// TwinCAT 3 PLC project LeakTesters
// ProgramVersion: 3.1.4024.0
// libraries:
//   Tc2_Standard, * (Beckhoff Automation GmbH)
//   Tc2_System, * (Beckhoff Automation GmbH)
//   Tc2_Utilities, * (Beckhoff Automation GmbH)
//   Tc3_EventLogger, * (Beckhoff Automation GmbH)
//   Tc3_Module, * (Beckhoff Automation GmbH)
//   VisuUserMgmt, * (System)
// project tree:
//   DUTs/ E_CameraJobChange.TcDUT, E_MachineState.TcDUT (not stored), E_StationState.TcDUT (not stored), ST_ActiveEventsHMI.TcDUT (not stored), ST_AlarmHistory.TcDUT (not stored), ST_Events.TcDUT (not stored), ST_HeightLimits.TcDUT, ST_HeightMeasurement2.TcDUT, ST_MachineStatusStruct.TcDUT (not stored), ST_MasterControlStruct.TcDUT (not stored), ST_MeasureStatistics.TcDUT (not stored), ST_Nest.TcDUT, ST_PartsInspection.TcDUT, ST_StandardStationStruct.TcDUT (not stored), ST_UserLogHMI.TcDUT (not stored)
//   DUTs/HeightMeasureFunction/ E_HeighttMeasureProcess.TcDUT
//   DUTs/IO/i28/ st_i28General_I_O.TcDUT (not stored), st_i28LasResult.TcDUT (not stored), st_i28LiveMeasurement.TcDUT (not stored)
//   DUTs/IO/ st_IS2802M.TcDUT, E_BoxDiag.TcDUT (not stored), E_BoxState.TcDUT (not stored), E_TerminalState.TcDUT (not stored), st_Box_Info.TcDUT (not stored), st_EL1809.TcDUT (not stored), st_EL2809.TcDUT (not stored), ST_DL_PN1.TcDUT, st_Terminal_Info.TcDUT (not stored)
//   GVLs/ GVL_Constants.TcGVL (not stored), GVL_HMI_GLOBAL.TcGVL, GVL_IO.TcGVL, GVL_MASTER.TcGVL, GVL_PERSIST.TcGVL
//   / PlcTask.TcTTO (not stored)
//   POUs/A_Master/ Main_Master.TcPOU, PRG_FaultHandling.TcPOU, PRG_MachineStatus.TcPOU, PRG_MasterCycle.TcPOU, PRG_MasterSystemTime.TcPOU (not stored), PRG_TerminBoxInfo.TcPOU (not stored)
//   POUs/B_HightTest/ PRG_Fault_HeightTest.TcPOU, PRG_HeightTest.TcPOU
//   POUs/C_LeakTest/ PRG_Fault_LeakTest.TcPOU, PRG_LeakTest.TcPOU, PRG_LeakTestEvents_Info.TcPOU
//   POUs/D_VisionTest/ PRG_Fault_VisionTest.TcPOU, PRG_VisionTest.TcPOU
//   POUs/E_HMI/ PRG_HMI.TcPOU
//   POUs/G_Utility/ FB_Alarms.TcPOU (not stored), FB_BoxInfo.TcPOU (not stored), FB_DayOfYear.TcPOU (not stored), FB_EventLog.TcPOU (not stored), FB_HeightMeasurement2.TcPOU, FB_Pulse.TcPOU (not stored), FB_TerminalInfo.TcPOU (not stored), FB_TimeControl.TcPOU (not stored), PRG_Puls.TcPOU (not stored)
//   POUs/ MAIN.TcPOU (not stored)
// real-time tasks:
//   TASK PlcTask: cycle T#10ms, priority 20, ADS port 350
// I/O:
//   DEVICE Device 1 (EtherCAT), AmsNetId 172.18.237.82.2.1
//     Term 9 (EK1100) [EK1100 EtherCAT Coupler (2A E-Bus)]
//       Term 10 (EL6070-0033) [EL6070-0033 1Ch. Licence key terminal, individual licences]
//       Term 11 (EL1809) [EL1809 16Ch. Dig. Input 24V, 3ms]
//       Term 12 (EL2809-0015) [EL2809-0015 16Ch. Dig. Output 24V DC, 0.35A, not short-circuit proof]
//       Term 13 (EL6631) [EL6631 PROFINET IO Controller]
//       Term 14 (EL9011) [EL9011 End Terminal]
//   DEVICE Device 2 (EL6631), AmsNetId 172.18.237.82.3.1
//     is2802 [Cognex Corp. In-Sight IS28XX Vision System IS28XX-XX]
//       modules: Term 1 (DAP Module), Term 2 (Acquisition Control), Term 3 (Acquisition Status), Term 4 (Inspection Control), Term 5 (Inspection Status), Term 6 (Command Control), Term 7 (ExternalEvent Control), Term 8 (User Data - 64 bytes), Term 9 (Results - 64 bytes)
//     i28 [Cincinnati Test Systems 1-port Device 00210]
//       modules: Term 10 (DAP Module), Term 11 (PLC Input), Term 12 (PLC Output  )
//     dl-pn1 [Keyence DL-PN1 PROFINET IO Device DL-PN1]
//       modules: Term 13 (DAP Module), Term 14 (DL-PN1), Term 15 (GT2-1.1), Term 16 (GT2-1.2), Term 17 (GT2-1.3), Term 18 (GT2-2)
// variable links:
//   LeakTesters/LeakTesters Instance <-> Device 1 (EtherCAT)/Term 9 (EK1100)/Term 10 (EL6070-0033)
//     PlcTask Inputs/GVL_IO.dwTerminalInfo[2].nTerminal_State <-> InfoData/State
//   LeakTesters/LeakTesters Instance <-> Device 1 (EtherCAT)/Term 9 (EK1100)/Term 11 (EL1809)
//     PlcTask Inputs/GVL_IO.dwTerminalInfo[3].nTerminal_State <-> InfoData/State
//     PlcTask Inputs/GVL_IO.dw_T02_EL1809.iCalmpClosed <-> Channel 1/Input
//     PlcTask Inputs/GVL_IO.dw_T02_EL1809.iPartPresent <-> Channel 2/Input
//   LeakTesters/LeakTesters Instance <-> Device 1 (EtherCAT)/Term 9 (EK1100)/Term 12 (EL2809-0015)
//     PlcTask Inputs/GVL_IO.dwTerminalInfo[4].nTerminal_State <-> InfoData/State
//     PlcTask Outputs/GVL_IO.dw_T03_EL2809.qEL2809_Ch3 <-> Channel 3/Output
//     PlcTask Outputs/GVL_IO.dw_T03_EL2809.qPassIndicatorGreen <-> Channel 1/Output
//     PlcTask Outputs/GVL_IO.dw_T03_EL2809.qRejectIndicatorRed <-> Channel 2/Output
//   LeakTesters/LeakTesters Instance <-> Device 1 (EtherCAT)/Term 9 (EK1100)/Term 13 (EL6631)
//     PlcTask Inputs/GVL_IO.dwTerminalInfo[5].nTerminal_State <-> InfoData/State
//   LeakTesters/LeakTesters Instance <-> Device 2 (EL6631)/dl-pn1
//     PlcTask Inputs/GVL_IO.dwBoxInfo[17].nPnIoBoxDiag <-> Inputs/PnIoBoxDiag
//     PlcTask Inputs/GVL_IO.dwBoxInfo[17].nPnIoBoxState <-> Inputs/PnIoBoxState
//     PlcTask Inputs/GVL_IO.dw_B08_DL_PN1.dldCurrValProp <-> API/Term 14 (DL-PN1)/Subterm 23 (DL-PN1 Device)/Inputs/Sensors Status/Current_Value_Property
//     PlcTask Inputs/GVL_IO.dw_B08_DL_PN1.dldErrorStt <-> API/Term 14 (DL-PN1)/Subterm 23 (DL-PN1 Device)/Inputs/Sensors Status/Error_Status
//     PlcTask Inputs/GVL_IO.dw_B08_DL_PN1.dldExtInpResp[1] <-> API/Term 14 (DL-PN1)/Subterm 23 (DL-PN1 Device)/Inputs/External Input Response/External_Input_Response_1
//     PlcTask Inputs/GVL_IO.dw_B08_DL_PN1.dldExtInpResp[2] <-> API/Term 14 (DL-PN1)/Subterm 23 (DL-PN1 Device)/Inputs/External Input Response/External_Input_Response_2
//     PlcTask Inputs/GVL_IO.dw_B08_DL_PN1.dldExtInpResp[3] <-> API/Term 14 (DL-PN1)/Subterm 23 (DL-PN1 Device)/Inputs/External Input Response/External_Input_Response_3
//     PlcTask Inputs/GVL_IO.dw_B08_DL_PN1.dldExtInpResp[4] <-> API/Term 14 (DL-PN1)/Subterm 23 (DL-PN1 Device)/Inputs/External Input Response/External_Input_Response_4
//     PlcTask Inputs/GVL_IO.dw_B08_DL_PN1.dldExtInpResp[5] <-> API/Term 14 (DL-PN1)/Subterm 23 (DL-PN1 Device)/Inputs/External Input Response/External_Input_Response_5
//     PlcTask Inputs/GVL_IO.dw_B08_DL_PN1.dldWarningStat <-> API/Term 14 (DL-PN1)/Subterm 23 (DL-PN1 Device)/Inputs/Sensors Status/Warning_Status
//     PlcTask Inputs/GVL_IO.dw_B08_DL_PN1.gt2_1_1CurrValInv <-> API/Term 15 (GT2-1.1)/Subterm 24 (GT2-***)/Inputs/Sensor Status/Current_Value_Invalid
//     PlcTask Inputs/GVL_IO.dw_B08_DL_PN1.gt2_1_2CurrValInv <-> API/Term 16 (GT2-1.2)/Subterm 25 (GT2-***)/Inputs/Sensor Status/Current_Value_Invalid
//     PlcTask Inputs/GVL_IO.dw_B08_DL_PN1.gt2_1_3CurrValInv <-> API/Term 17 (GT2-1.3)/Subterm 26 (GT2-***)/Inputs/Sensor Status/Current_Value_Invalid
//     PlcTask Inputs/GVL_IO.dw_B08_DL_PN1.gt2_1_1CurrValOvrR <-> API/Term 15 (GT2-1.1)/Subterm 24 (GT2-***)/Inputs/Sensor Status/Current_Value_Over_Range
//     PlcTask Inputs/GVL_IO.dw_B08_DL_PN1.gt2_1_2CurrValOvrR <-> API/Term 16 (GT2-1.2)/Subterm 25 (GT2-***)/Inputs/Sensor Status/Current_Value_Over_Range
//     PlcTask Inputs/GVL_IO.dw_B08_DL_PN1.gt2_1_3CurrValOvrR <-> API/Term 17 (GT2-1.3)/Subterm 26 (GT2-***)/Inputs/Sensor Status/Current_Value_Over_Range
//     PlcTask Inputs/GVL_IO.dw_B08_DL_PN1.gt2_1_1CurrValUndR <-> API/Term 15 (GT2-1.1)/Subterm 24 (GT2-***)/Inputs/Sensor Status/Current_Value_Under_Range
//     PlcTask Inputs/GVL_IO.dw_B08_DL_PN1.gt2_1_2CurrValUndR <-> API/Term 16 (GT2-1.2)/Subterm 25 (GT2-***)/Inputs/Sensor Status/Current_Value_Under_Range
//     PlcTask Inputs/GVL_IO.dw_B08_DL_PN1.gt2_1_3CurrValUndR <-> API/Term 17 (GT2-1.3)/Subterm 26 (GT2-***)/Inputs/Sensor Status/Current_Value_Under_Range
//     PlcTask Inputs/GVL_IO.dw_B08_DL_PN1.gt2_1_1CurrentValue <-> API/Term 15 (GT2-1.1)/Subterm 24 (GT2-***)/Inputs/Current Value
//     PlcTask Inputs/GVL_IO.dw_B08_DL_PN1.gt2_1_2CurrentValue <-> API/Term 16 (GT2-1.2)/Subterm 25 (GT2-***)/Inputs/Current Value
//     PlcTask Inputs/GVL_IO.dw_B08_DL_PN1.gt2_1_3CurrentValue <-> API/Term 17 (GT2-1.3)/Subterm 26 (GT2-***)/Inputs/Current Value
//     PlcTask Inputs/GVL_IO.dw_B08_DL_PN1.gt2_1_1ErrorStat <-> API/Term 15 (GT2-1.1)/Subterm 24 (GT2-***)/Inputs/Sensor Status/Error_Status
//     PlcTask Inputs/GVL_IO.dw_B08_DL_PN1.gt2_1_2ErrorStat <-> API/Term 16 (GT2-1.2)/Subterm 25 (GT2-***)/Inputs/Sensor Status/Error_Status
//     PlcTask Inputs/GVL_IO.dw_B08_DL_PN1.gt2_1_3ErrorStat <-> API/Term 17 (GT2-1.3)/Subterm 26 (GT2-***)/Inputs/Sensor Status/Error_Status
//     PlcTask Inputs/GVL_IO.dw_B08_DL_PN1.gt2_1_1ExtInpRes[1] <-> API/Term 15 (GT2-1.1)/Subterm 24 (GT2-***)/Inputs/External Input Response/External_Input_Response_1
//     PlcTask Inputs/GVL_IO.dw_B08_DL_PN1.gt2_1_1ExtInpRes[2] <-> API/Term 15 (GT2-1.1)/Subterm 24 (GT2-***)/Inputs/External Input Response/External_Input_Response_2
//     PlcTask Inputs/GVL_IO.dw_B08_DL_PN1.gt2_1_1ExtInpRes[3] <-> API/Term 15 (GT2-1.1)/Subterm 24 (GT2-***)/Inputs/External Input Response/External_Input_Response_3
//     PlcTask Inputs/GVL_IO.dw_B08_DL_PN1.gt2_1_1ExtInpRes[4] <-> API/Term 15 (GT2-1.1)/Subterm 24 (GT2-***)/Inputs/External Input Response/External_Input_Response_4
//     PlcTask Inputs/GVL_IO.dw_B08_DL_PN1.gt2_1_1ExtInpRes[5] <-> API/Term 15 (GT2-1.1)/Subterm 24 (GT2-***)/Inputs/External Input Response/External_Input_Response_5
//     PlcTask Inputs/GVL_IO.dw_B08_DL_PN1.gt2_1_2ExtInpRes[1] <-> API/Term 16 (GT2-1.2)/Subterm 25 (GT2-***)/Inputs/External Input Response/External_Input_Response_1
//     PlcTask Inputs/GVL_IO.dw_B08_DL_PN1.gt2_1_2ExtInpRes[2] <-> API/Term 16 (GT2-1.2)/Subterm 25 (GT2-***)/Inputs/External Input Response/External_Input_Response_2
//     PlcTask Inputs/GVL_IO.dw_B08_DL_PN1.gt2_1_2ExtInpRes[3] <-> API/Term 16 (GT2-1.2)/Subterm 25 (GT2-***)/Inputs/External Input Response/External_Input_Response_3
//     PlcTask Inputs/GVL_IO.dw_B08_DL_PN1.gt2_1_2ExtInpRes[4] <-> API/Term 16 (GT2-1.2)/Subterm 25 (GT2-***)/Inputs/External Input Response/External_Input_Response_4
//     PlcTask Inputs/GVL_IO.dw_B08_DL_PN1.gt2_1_2ExtInpRes[5] <-> API/Term 16 (GT2-1.2)/Subterm 25 (GT2-***)/Inputs/External Input Response/External_Input_Response_5
//     PlcTask Inputs/GVL_IO.dw_B08_DL_PN1.gt2_1_3ExtInpRes[1] <-> API/Term 17 (GT2-1.3)/Subterm 26 (GT2-***)/Inputs/External Input Response/External_Input_Response_1
//     PlcTask Inputs/GVL_IO.dw_B08_DL_PN1.gt2_1_3ExtInpRes[2] <-> API/Term 17 (GT2-1.3)/Subterm 26 (GT2-***)/Inputs/External Input Response/External_Input_Response_2
//     PlcTask Inputs/GVL_IO.dw_B08_DL_PN1.gt2_1_3ExtInpRes[3] <-> API/Term 17 (GT2-1.3)/Subterm 26 (GT2-***)/Inputs/External Input Response/External_Input_Response_3
//     PlcTask Inputs/GVL_IO.dw_B08_DL_PN1.gt2_1_3ExtInpRes[4] <-> API/Term 17 (GT2-1.3)/Subterm 26 (GT2-***)/Inputs/External Input Response/External_Input_Response_4
//     PlcTask Inputs/GVL_IO.dw_B08_DL_PN1.gt2_1_3ExtInpRes[5] <-> API/Term 17 (GT2-1.3)/Subterm 26 (GT2-***)/Inputs/External Input Response/External_Input_Response_5
//     PlcTask Inputs/GVL_IO.dw_B08_DL_PN1.gt2_1_1Output[1] <-> API/Term 15 (GT2-1.1)/Subterm 24 (GT2-***)/Inputs/Sensor Outputs/Output_1
//     PlcTask Inputs/GVL_IO.dw_B08_DL_PN1.gt2_1_1Output[2] <-> API/Term 15 (GT2-1.1)/Subterm 24 (GT2-***)/Inputs/Sensor Outputs/Output_2
//     PlcTask Inputs/GVL_IO.dw_B08_DL_PN1.gt2_1_1Output[3] <-> API/Term 15 (GT2-1.1)/Subterm 24 (GT2-***)/Inputs/Sensor Outputs/Output_3
//     PlcTask Inputs/GVL_IO.dw_B08_DL_PN1.gt2_1_1Output[4] <-> API/Term 15 (GT2-1.1)/Subterm 24 (GT2-***)/Inputs/Sensor Outputs/Output_4
//     PlcTask Inputs/GVL_IO.dw_B08_DL_PN1.gt2_1_1Output[5] <-> API/Term 15 (GT2-1.1)/Subterm 24 (GT2-***)/Inputs/Sensor Outputs/Output_5
//     PlcTask Inputs/GVL_IO.dw_B08_DL_PN1.gt2_1_2Output[1] <-> API/Term 16 (GT2-1.2)/Subterm 25 (GT2-***)/Inputs/Sensor Outputs/Output_1
//     PlcTask Inputs/GVL_IO.dw_B08_DL_PN1.gt2_1_2Output[2] <-> API/Term 16 (GT2-1.2)/Subterm 25 (GT2-***)/Inputs/Sensor Outputs/Output_2
//     PlcTask Inputs/GVL_IO.dw_B08_DL_PN1.gt2_1_2Output[3] <-> API/Term 16 (GT2-1.2)/Subterm 25 (GT2-***)/Inputs/Sensor Outputs/Output_3
//     PlcTask Inputs/GVL_IO.dw_B08_DL_PN1.gt2_1_2Output[4] <-> API/Term 16 (GT2-1.2)/Subterm 25 (GT2-***)/Inputs/Sensor Outputs/Output_4
//     PlcTask Inputs/GVL_IO.dw_B08_DL_PN1.gt2_1_2Output[5] <-> API/Term 16 (GT2-1.2)/Subterm 25 (GT2-***)/Inputs/Sensor Outputs/Output_5
//     PlcTask Inputs/GVL_IO.dw_B08_DL_PN1.gt2_1_3Output[1] <-> API/Term 17 (GT2-1.3)/Subterm 26 (GT2-***)/Inputs/Sensor Outputs/Output_1
//     PlcTask Inputs/GVL_IO.dw_B08_DL_PN1.gt2_1_3Output[2] <-> API/Term 17 (GT2-1.3)/Subterm 26 (GT2-***)/Inputs/Sensor Outputs/Output_2
//     PlcTask Inputs/GVL_IO.dw_B08_DL_PN1.gt2_1_3Output[3] <-> API/Term 17 (GT2-1.3)/Subterm 26 (GT2-***)/Inputs/Sensor Outputs/Output_3
//     PlcTask Inputs/GVL_IO.dw_B08_DL_PN1.gt2_1_3Output[4] <-> API/Term 17 (GT2-1.3)/Subterm 26 (GT2-***)/Inputs/Sensor Outputs/Output_4
//     PlcTask Inputs/GVL_IO.dw_B08_DL_PN1.gt2_1_3Output[5] <-> API/Term 17 (GT2-1.3)/Subterm 26 (GT2-***)/Inputs/Sensor Outputs/Output_5
//     PlcTask Inputs/GVL_IO.dw_B08_DL_PN1.gt2_1_1WarningStat <-> API/Term 15 (GT2-1.1)/Subterm 24 (GT2-***)/Inputs/Sensor Status/Warning_Status
//     PlcTask Inputs/GVL_IO.dw_B08_DL_PN1.gt2_1_2WarningStat <-> API/Term 16 (GT2-1.2)/Subterm 25 (GT2-***)/Inputs/Sensor Status/Warning_Status
//     PlcTask Inputs/GVL_IO.dw_B08_DL_PN1.gt2_1_3WarningStat <-> API/Term 17 (GT2-1.3)/Subterm 26 (GT2-***)/Inputs/Sensor Status/Warning_Status
//     PlcTask Inputs/GVL_IO.dw_B08_DL_PN1.gt2_2CurrValInv <-> API/Term 18 (GT2-2)/Subterm 27 (GT2-***)/Inputs/Sensor Status/Current_Value_Invalid
//     PlcTask Inputs/GVL_IO.dw_B08_DL_PN1.gt2_2CurrValOvrR <-> API/Term 18 (GT2-2)/Subterm 27 (GT2-***)/Inputs/Sensor Status/Current_Value_Over_Range
//     PlcTask Inputs/GVL_IO.dw_B08_DL_PN1.gt2_2CurrValUndR <-> API/Term 18 (GT2-2)/Subterm 27 (GT2-***)/Inputs/Sensor Status/Current_Value_Under_Range
//     PlcTask Inputs/GVL_IO.dw_B08_DL_PN1.gt2_2CurrentValue <-> API/Term 18 (GT2-2)/Subterm 27 (GT2-***)/Inputs/Current Value
//     PlcTask Inputs/GVL_IO.dw_B08_DL_PN1.gt2_2ErrorStat <-> API/Term 18 (GT2-2)/Subterm 27 (GT2-***)/Inputs/Sensor Status/Error_Status
//     PlcTask Inputs/GVL_IO.dw_B08_DL_PN1.gt2_2ExtInpRes[1] <-> API/Term 18 (GT2-2)/Subterm 27 (GT2-***)/Inputs/External Input Response/External_Input_Response_1
//     PlcTask Inputs/GVL_IO.dw_B08_DL_PN1.gt2_2ExtInpRes[2] <-> API/Term 18 (GT2-2)/Subterm 27 (GT2-***)/Inputs/External Input Response/External_Input_Response_2
//     PlcTask Inputs/GVL_IO.dw_B08_DL_PN1.gt2_2ExtInpRes[3] <-> API/Term 18 (GT2-2)/Subterm 27 (GT2-***)/Inputs/External Input Response/External_Input_Response_3
//     PlcTask Inputs/GVL_IO.dw_B08_DL_PN1.gt2_2ExtInpRes[4] <-> API/Term 18 (GT2-2)/Subterm 27 (GT2-***)/Inputs/External Input Response/External_Input_Response_4
//     PlcTask Inputs/GVL_IO.dw_B08_DL_PN1.gt2_2ExtInpRes[5] <-> API/Term 18 (GT2-2)/Subterm 27 (GT2-***)/Inputs/External Input Response/External_Input_Response_5
//     PlcTask Inputs/GVL_IO.dw_B08_DL_PN1.gt2_2Output[1] <-> API/Term 18 (GT2-2)/Subterm 27 (GT2-***)/Inputs/Sensor Outputs/Output_1
//     PlcTask Inputs/GVL_IO.dw_B08_DL_PN1.gt2_2Output[2] <-> API/Term 18 (GT2-2)/Subterm 27 (GT2-***)/Inputs/Sensor Outputs/Output_2
//     PlcTask Inputs/GVL_IO.dw_B08_DL_PN1.gt2_2Output[3] <-> API/Term 18 (GT2-2)/Subterm 27 (GT2-***)/Inputs/Sensor Outputs/Output_3
//     PlcTask Inputs/GVL_IO.dw_B08_DL_PN1.gt2_2Output[4] <-> API/Term 18 (GT2-2)/Subterm 27 (GT2-***)/Inputs/Sensor Outputs/Output_4
//     PlcTask Inputs/GVL_IO.dw_B08_DL_PN1.gt2_2Output[5] <-> API/Term 18 (GT2-2)/Subterm 27 (GT2-***)/Inputs/Sensor Outputs/Output_5
//     PlcTask Inputs/GVL_IO.dw_B08_DL_PN1.gt2_2WarningStat <-> API/Term 18 (GT2-2)/Subterm 27 (GT2-***)/Inputs/Sensor Status/Warning_Status
//     PlcTask Outputs/GVL_IO.dw_B08_DL_PN1.dldExtInpRespOut[1] <-> API/Term 14 (DL-PN1)/Subterm 23 (DL-PN1 Device)/Outputs/External Input Requests/External_Input_Request_1
//     PlcTask Outputs/GVL_IO.dw_B08_DL_PN1.dldExtInpRespOut[2] <-> API/Term 14 (DL-PN1)/Subterm 23 (DL-PN1 Device)/Outputs/External Input Requests/External_Input_Request_2
//     PlcTask Outputs/GVL_IO.dw_B08_DL_PN1.dldExtInpRespOut[3] <-> API/Term 14 (DL-PN1)/Subterm 23 (DL-PN1 Device)/Outputs/External Input Requests/External_Input_Request_3
//     PlcTask Outputs/GVL_IO.dw_B08_DL_PN1.dldExtInpRespOut[4] <-> API/Term 14 (DL-PN1)/Subterm 23 (DL-PN1 Device)/Outputs/External Input Requests/External_Input_Request_4
//     PlcTask Outputs/GVL_IO.dw_B08_DL_PN1.dldExtInpRespOut[5] <-> API/Term 14 (DL-PN1)/Subterm 23 (DL-PN1 Device)/Outputs/External Input Requests/External_Input_Request_5
//     PlcTask Outputs/GVL_IO.dw_B08_DL_PN1.gt2_1_1ExtInpResOut[1] <-> API/Term 15 (GT2-1.1)/Subterm 24 (GT2-***)/Outputs/External Input Requests/External_Input_Request_1
//     PlcTask Outputs/GVL_IO.dw_B08_DL_PN1.gt2_1_1ExtInpResOut[2] <-> API/Term 15 (GT2-1.1)/Subterm 24 (GT2-***)/Outputs/External Input Requests/External_Input_Request_2
//     PlcTask Outputs/GVL_IO.dw_B08_DL_PN1.gt2_1_1ExtInpResOut[3] <-> API/Term 15 (GT2-1.1)/Subterm 24 (GT2-***)/Outputs/External Input Requests/External_Input_Request_3
//     PlcTask Outputs/GVL_IO.dw_B08_DL_PN1.gt2_1_1ExtInpResOut[4] <-> API/Term 15 (GT2-1.1)/Subterm 24 (GT2-***)/Outputs/External Input Requests/External_Input_Request_4
//     PlcTask Outputs/GVL_IO.dw_B08_DL_PN1.gt2_1_1ExtInpResOut[5] <-> API/Term 15 (GT2-1.1)/Subterm 24 (GT2-***)/Outputs/External Input Requests/External_Input_Request_5
//     PlcTask Outputs/GVL_IO.dw_B08_DL_PN1.gt2_1_2ExtInpResOut[1] <-> API/Term 16 (GT2-1.2)/Subterm 25 (GT2-***)/Outputs/External Input Requests/External_Input_Request_1
//     PlcTask Outputs/GVL_IO.dw_B08_DL_PN1.gt2_1_2ExtInpResOut[2] <-> API/Term 16 (GT2-1.2)/Subterm 25 (GT2-***)/Outputs/External Input Requests/External_Input_Request_2
//     PlcTask Outputs/GVL_IO.dw_B08_DL_PN1.gt2_1_2ExtInpResOut[3] <-> API/Term 16 (GT2-1.2)/Subterm 25 (GT2-***)/Outputs/External Input Requests/External_Input_Request_3
//     PlcTask Outputs/GVL_IO.dw_B08_DL_PN1.gt2_1_2ExtInpResOut[4] <-> API/Term 16 (GT2-1.2)/Subterm 25 (GT2-***)/Outputs/External Input Requests/External_Input_Request_4
//     PlcTask Outputs/GVL_IO.dw_B08_DL_PN1.gt2_1_2ExtInpResOut[5] <-> API/Term 16 (GT2-1.2)/Subterm 25 (GT2-***)/Outputs/External Input Requests/External_Input_Request_5
//     PlcTask Outputs/GVL_IO.dw_B08_DL_PN1.gt2_1_3ExtInpResOut[1] <-> API/Term 17 (GT2-1.3)/Subterm 26 (GT2-***)/Outputs/External Input Requests/External_Input_Request_1
//     PlcTask Outputs/GVL_IO.dw_B08_DL_PN1.gt2_1_3ExtInpResOut[2] <-> API/Term 17 (GT2-1.3)/Subterm 26 (GT2-***)/Outputs/External Input Requests/External_Input_Request_2
//     PlcTask Outputs/GVL_IO.dw_B08_DL_PN1.gt2_1_3ExtInpResOut[3] <-> API/Term 17 (GT2-1.3)/Subterm 26 (GT2-***)/Outputs/External Input Requests/External_Input_Request_3
//     PlcTask Outputs/GVL_IO.dw_B08_DL_PN1.gt2_1_3ExtInpResOut[4] <-> API/Term 17 (GT2-1.3)/Subterm 26 (GT2-***)/Outputs/External Input Requests/External_Input_Request_4
//     PlcTask Outputs/GVL_IO.dw_B08_DL_PN1.gt2_1_3ExtInpResOut[5] <-> API/Term 17 (GT2-1.3)/Subterm 26 (GT2-***)/Outputs/External Input Requests/External_Input_Request_5
//     PlcTask Outputs/GVL_IO.dw_B08_DL_PN1.gt2_2ExtInpResOut[1] <-> API/Term 18 (GT2-2)/Subterm 27 (GT2-***)/Outputs/External Input Requests/External_Input_Request_1
//     PlcTask Outputs/GVL_IO.dw_B08_DL_PN1.gt2_2ExtInpResOut[2] <-> API/Term 18 (GT2-2)/Subterm 27 (GT2-***)/Outputs/External Input Requests/External_Input_Request_2
//     PlcTask Outputs/GVL_IO.dw_B08_DL_PN1.gt2_2ExtInpResOut[3] <-> API/Term 18 (GT2-2)/Subterm 27 (GT2-***)/Outputs/External Input Requests/External_Input_Request_3
//     PlcTask Outputs/GVL_IO.dw_B08_DL_PN1.gt2_2ExtInpResOut[4] <-> API/Term 18 (GT2-2)/Subterm 27 (GT2-***)/Outputs/External Input Requests/External_Input_Request_4
//     PlcTask Outputs/GVL_IO.dw_B08_DL_PN1.gt2_2ExtInpResOut[5] <-> API/Term 18 (GT2-2)/Subterm 27 (GT2-***)/Outputs/External Input Requests/External_Input_Request_5
//   LeakTesters/LeakTesters Instance <-> Device 2 (EL6631)/i28
//     PlcTask Inputs/GVL_IO.dwBoxInfo[16].nPnIoBoxDiag <-> Inputs/PnIoBoxDiag
//     PlcTask Inputs/GVL_IO.dwBoxInfo[16].nPnIoBoxState <-> Inputs/PnIoBoxState
//     PlcTask Inputs/GVL_IO.dw_B07_i28General_I_O.bInput1 <-> API/Term 11 (PLC Input)/Subterm 15 (Instrument Status)/Inputs/Instrument Status/User_Configurable_Input_1
//     PlcTask Inputs/GVL_IO.dw_B07_i28General_I_O.bInput10 <-> API/Term 11 (PLC Input)/Subterm 15 (Instrument Status)/Inputs/Instrument Status/User_Configurable_Input_10
//     PlcTask Inputs/GVL_IO.dw_B07_i28General_I_O.bInput11 <-> API/Term 11 (PLC Input)/Subterm 15 (Instrument Status)/Inputs/Instrument Status/User_Configurable_Input_11
//     PlcTask Inputs/GVL_IO.dw_B07_i28General_I_O.bInput12 <-> API/Term 11 (PLC Input)/Subterm 15 (Instrument Status)/Inputs/Instrument Status/User_Configurable_Input_12
//     PlcTask Inputs/GVL_IO.dw_B07_i28General_I_O.bInput13 <-> API/Term 11 (PLC Input)/Subterm 15 (Instrument Status)/Inputs/Instrument Status/User_Configurable_Input_13
//     PlcTask Inputs/GVL_IO.dw_B07_i28General_I_O.bInput14 <-> API/Term 11 (PLC Input)/Subterm 15 (Instrument Status)/Inputs/Instrument Status/User_Configurable_Input_14
//     PlcTask Inputs/GVL_IO.dw_B07_i28General_I_O.bInput15 <-> API/Term 11 (PLC Input)/Subterm 15 (Instrument Status)/Inputs/Instrument Status/User_Configurable_Input_15
//     PlcTask Inputs/GVL_IO.dw_B07_i28General_I_O.bInput16 <-> API/Term 11 (PLC Input)/Subterm 15 (Instrument Status)/Inputs/Instrument Status/User_Configurable_Input_16
//     PlcTask Inputs/GVL_IO.dw_B07_i28General_I_O.bInput2 <-> API/Term 11 (PLC Input)/Subterm 15 (Instrument Status)/Inputs/Instrument Status/User_Configurable_Input_2
//     PlcTask Inputs/GVL_IO.dw_B07_i28General_I_O.bInput3 <-> API/Term 11 (PLC Input)/Subterm 15 (Instrument Status)/Inputs/Instrument Status/User_Configurable_Input_3
//     PlcTask Inputs/GVL_IO.dw_B07_i28General_I_O.bInput4 <-> API/Term 11 (PLC Input)/Subterm 15 (Instrument Status)/Inputs/Instrument Status/User_Configurable_Input_4
//     PlcTask Inputs/GVL_IO.dw_B07_i28General_I_O.bInput5 <-> API/Term 11 (PLC Input)/Subterm 15 (Instrument Status)/Inputs/Instrument Status/User_Configurable_Input_5
//     PlcTask Inputs/GVL_IO.dw_B07_i28General_I_O.bInput6 <-> API/Term 11 (PLC Input)/Subterm 15 (Instrument Status)/Inputs/Instrument Status/User_Configurable_Input_6
//     PlcTask Inputs/GVL_IO.dw_B07_i28General_I_O.bInput7 <-> API/Term 11 (PLC Input)/Subterm 15 (Instrument Status)/Inputs/Instrument Status/User_Configurable_Input_7
//     PlcTask Inputs/GVL_IO.dw_B07_i28General_I_O.bInput8 <-> API/Term 11 (PLC Input)/Subterm 15 (Instrument Status)/Inputs/Instrument Status/User_Configurable_Input_8
//     PlcTask Inputs/GVL_IO.dw_B07_i28General_I_O.bInput9 <-> API/Term 11 (PLC Input)/Subterm 15 (Instrument Status)/Inputs/Instrument Status/User_Configurable_Input_9
//     PlcTask Inputs/GVL_IO.dw_B07_i28General_I_O.bInstrumentReady <-> API/Term 11 (PLC Input)/Subterm 15 (Instrument Status)/Inputs/Instrument Status/Instrument_Ready
//     PlcTask Inputs/GVL_IO.dw_B07_i28General_I_O.bMalfunction <-> API/Term 11 (PLC Input)/Subterm 15 (Instrument Status)/Inputs/Instrument Status/Malfunction
//     PlcTask Inputs/GVL_IO.dw_B07_i28General_I_O.bProgramAccept <-> API/Term 11 (PLC Input)/Subterm 15 (Instrument Status)/Inputs/Instrument Status/Program_Accept
//     PlcTask Inputs/GVL_IO.dw_B07_i28General_I_O.bProgramReject <-> API/Term 11 (PLC Input)/Subterm 15 (Instrument Status)/Inputs/Instrument Status/Program_Reject
//     PlcTask Inputs/GVL_IO.dw_B07_i28General_I_O.bTestActiveLiveData <-> API/Term 11 (PLC Input)/Subterm 15 (Instrument Status)/Inputs/Instrument Status/Test_Active_Live_Data
//     PlcTask Inputs/GVL_IO.dw_B07_i28General_I_O.nCurrentProgramNumber <-> API/Term 11 (PLC Input)/Subterm 15 (Instrument Status)/Inputs/Current_Program Number
//     PlcTask Inputs/GVL_IO.dw_B07_i28LastResult.ibTestEvaluation0 <-> API/Term 11 (PLC Input)/Subterm 17 (Last test result)/Inputs/Test Evaluation Code/Test_Evaluation_Code_Bit_0
//     PlcTask Inputs/GVL_IO.dw_B07_i28LastResult.ibTestEvaluation1 <-> API/Term 11 (PLC Input)/Subterm 17 (Last test result)/Inputs/Test Evaluation Code/Test_Evaluation_Code_Bit_1
//     PlcTask Inputs/GVL_IO.dw_B07_i28LastResult.ibTestEvaluation2 <-> API/Term 11 (PLC Input)/Subterm 17 (Last test result)/Inputs/Test Evaluation Code/Test_Evaluation_Code_Bit_2
//     PlcTask Inputs/GVL_IO.dw_B07_i28LastResult.ibTestEvaluation3 <-> API/Term 11 (PLC Input)/Subterm 17 (Last test result)/Inputs/Test Evaluation Code/Test_Evaluation_Code_Bit_3
//     PlcTask Inputs/GVL_IO.dw_B07_i28LastResult.inChannelNumber <-> API/Term 11 (PLC Input)/Subterm 17 (Last test result)/Inputs/Channel Number
//     PlcTask Inputs/GVL_IO.dw_B07_i28LastResult.inMeasurement1 <-> API/Term 11 (PLC Input)/Subterm 17 (Last test result)/Inputs/Result Measurement 1
//     PlcTask Inputs/GVL_IO.dw_B07_i28LastResult.inMeasurement2 <-> API/Term 11 (PLC Input)/Subterm 17 (Last test result)/Inputs/Result Measurement 2
//     PlcTask Inputs/GVL_IO.dw_B07_i28LastResult.inPartEvaluation <-> API/Term 11 (PLC Input)/Subterm 17 (Last test result)/Inputs/Part Evaluation Code
//     PlcTask Inputs/GVL_IO.dw_B07_i28LastResult.inPrecisionCode <-> API/Term 11 (PLC Input)/Subterm 17 (Last test result)/Inputs/Precision Code
//     PlcTask Inputs/GVL_IO.dw_B07_i28LastResult.inProgramNumber <-> API/Term 11 (PLC Input)/Subterm 17 (Last test result)/Inputs/Program Number
//     PlcTask Inputs/GVL_IO.dw_B07_i28LastResult.inTestPort <-> API/Term 11 (PLC Input)/Subterm 17 (Last test result)/Inputs/Test Port
//     PlcTask Inputs/GVL_IO.dw_B07_i28LastResult.inTestType <-> API/Term 11 (PLC Input)/Subterm 17 (Last test result)/Inputs/Test Type Code
//     PlcTask Inputs/GVL_IO.dw_B07_i28LastResult.inUniqueID <-> API/Term 11 (PLC Input)/Subterm 17 (Last test result)/Inputs/Unique ID
//     PlcTask Inputs/GVL_IO.dw_B07_i28LastResult.inUnitCode1 <-> API/Term 11 (PLC Input)/Subterm 17 (Last test result)/Inputs/Unit Code[0]
//     PlcTask Inputs/GVL_IO.dw_B07_i28LastResult.inUnitCode2 <-> API/Term 11 (PLC Input)/Subterm 17 (Last test result)/Inputs/Unit Code[1]
//     PlcTask Inputs/GVL_IO.dw_B07_i28LastResult.inVariableCode1 <-> API/Term 11 (PLC Input)/Subterm 17 (Last test result)/Inputs/Variable Code[0]
//     PlcTask Inputs/GVL_IO.dw_B07_i28LastResult.inVariableCode2 <-> API/Term 11 (PLC Input)/Subterm 17 (Last test result)/Inputs/Variable Code[1]
//     PlcTask Inputs/GVL_IO.dw_B07_i28LiveMeasurement.inCurrentProgramNumber <-> API/Term 11 (PLC Input)/Subterm 16 (Live Measurement Data)/Inputs/Current Program Number
//     PlcTask Inputs/GVL_IO.dw_B07_i28LiveMeasurement.inMeasurement1 <-> API/Term 11 (PLC Input)/Subterm 16 (Live Measurement Data)/Inputs/Measurement 1 (Timer)
//     PlcTask Inputs/GVL_IO.dw_B07_i28LiveMeasurement.inMeasurement2 <-> API/Term 11 (PLC Input)/Subterm 16 (Live Measurement Data)/Inputs/Measurement 2 (Pressure)
//     PlcTask Inputs/GVL_IO.dw_B07_i28LiveMeasurement.inMeasurement3 <-> API/Term 11 (PLC Input)/Subterm 16 (Live Measurement Data)/Inputs/Measurement 3 (Pressure Loss/Rate)
//     PlcTask Inputs/GVL_IO.dw_B07_i28LiveMeasurement.inMeasurement4 <-> API/Term 11 (PLC Input)/Subterm 16 (Live Measurement Data)/Inputs/Measurement 4 (Flow/Leak)
//     PlcTask Inputs/GVL_IO.dw_B07_i28LiveMeasurement.inPrecisionCode1 <-> API/Term 11 (PLC Input)/Subterm 16 (Live Measurement Data)/Inputs/Precision Code[0]
//     PlcTask Inputs/GVL_IO.dw_B07_i28LiveMeasurement.inPrecisionCode2 <-> API/Term 11 (PLC Input)/Subterm 16 (Live Measurement Data)/Inputs/Precision Code[1]
//     PlcTask Inputs/GVL_IO.dw_B07_i28LiveMeasurement.inPrecisionCode3 <-> API/Term 11 (PLC Input)/Subterm 16 (Live Measurement Data)/Inputs/Precision Code[2]
//     PlcTask Inputs/GVL_IO.dw_B07_i28LiveMeasurement.inPrecisionCode4 <-> API/Term 11 (PLC Input)/Subterm 16 (Live Measurement Data)/Inputs/Precision Code[3]
//     PlcTask Inputs/GVL_IO.dw_B07_i28LiveMeasurement.inSegmentCode <-> API/Term 11 (PLC Input)/Subterm 16 (Live Measurement Data)/Inputs/Segment Code
//     PlcTask Inputs/GVL_IO.dw_B07_i28LiveMeasurement.inUniqueID <-> API/Term 11 (PLC Input)/Subterm 16 (Live Measurement Data)/Inputs/Unique ID
//     PlcTask Inputs/GVL_IO.dw_B07_i28LiveMeasurement.inUnitCode1 <-> API/Term 11 (PLC Input)/Subterm 16 (Live Measurement Data)/Inputs/Unit Code[0]
//     PlcTask Inputs/GVL_IO.dw_B07_i28LiveMeasurement.inUnitCode2 <-> API/Term 11 (PLC Input)/Subterm 16 (Live Measurement Data)/Inputs/Unit Code[1]
//     PlcTask Inputs/GVL_IO.dw_B07_i28LiveMeasurement.inUnitCode3 <-> API/Term 11 (PLC Input)/Subterm 16 (Live Measurement Data)/Inputs/Unit Code[2]
//     PlcTask Inputs/GVL_IO.dw_B07_i28LiveMeasurement.inUnitCode4 <-> API/Term 11 (PLC Input)/Subterm 16 (Live Measurement Data)/Inputs/Unit Code[3]
//     PlcTask Inputs/GVL_IO.dw_B07_i28LiveMeasurement.inVariableCode1 <-> API/Term 11 (PLC Input)/Subterm 16 (Live Measurement Data)/Inputs/Variable Code[0]
//     PlcTask Inputs/GVL_IO.dw_B07_i28LiveMeasurement.inVariableCode2 <-> API/Term 11 (PLC Input)/Subterm 16 (Live Measurement Data)/Inputs/Variable Code[1]
//     PlcTask Inputs/GVL_IO.dw_B07_i28LiveMeasurement.inVariableCode3 <-> API/Term 11 (PLC Input)/Subterm 16 (Live Measurement Data)/Inputs/Variable Code[2]
//     PlcTask Inputs/GVL_IO.dw_B07_i28LiveMeasurement.inVariableCode4 <-> API/Term 11 (PLC Input)/Subterm 16 (Live Measurement Data)/Inputs/Variable Code[3]
//     PlcTask Outputs/GVL_IO.dw_B07_i28General_I_O.bChangeProgram <-> API/Term 12 (PLC Output  )/Subterm 18 (Instrument Control )/Outputs/Instrument Control/Change_Program
//     PlcTask Outputs/GVL_IO.dw_B07_i28General_I_O.bOutput1 <-> API/Term 12 (PLC Output  )/Subterm 18 (Instrument Control )/Outputs/Instrument Control/User_Configurable_Output_1
//     PlcTask Outputs/GVL_IO.dw_B07_i28General_I_O.bOutput10 <-> API/Term 12 (PLC Output  )/Subterm 18 (Instrument Control )/Outputs/Instrument Control/User_Configurable_Output_10
//     PlcTask Outputs/GVL_IO.dw_B07_i28General_I_O.bOutput11 <-> API/Term 12 (PLC Output  )/Subterm 18 (Instrument Control )/Outputs/Instrument Control/User_Configurable_Output_11
//     PlcTask Outputs/GVL_IO.dw_B07_i28General_I_O.bOutput12 <-> API/Term 12 (PLC Output  )/Subterm 18 (Instrument Control )/Outputs/Instrument Control/User_Configurable_Output_12
//     PlcTask Outputs/GVL_IO.dw_B07_i28General_I_O.bOutput13 <-> API/Term 12 (PLC Output  )/Subterm 18 (Instrument Control )/Outputs/Instrument Control/User_Configurable_Output_13
//     PlcTask Outputs/GVL_IO.dw_B07_i28General_I_O.bOutput14 <-> API/Term 12 (PLC Output  )/Subterm 18 (Instrument Control )/Outputs/Instrument Control/User_Configurable_Output_14
//     PlcTask Outputs/GVL_IO.dw_B07_i28General_I_O.bOutput15 <-> API/Term 12 (PLC Output  )/Subterm 18 (Instrument Control )/Outputs/Instrument Control/User_Configurable_Output_15
//     PlcTask Outputs/GVL_IO.dw_B07_i28General_I_O.bOutput16 <-> API/Term 12 (PLC Output  )/Subterm 18 (Instrument Control )/Outputs/Instrument Control/User_Configurable_Output_16
//     PlcTask Outputs/GVL_IO.dw_B07_i28General_I_O.bOutput2 <-> API/Term 12 (PLC Output  )/Subterm 18 (Instrument Control )/Outputs/Instrument Control/User_Configurable_Output_2
//     PlcTask Outputs/GVL_IO.dw_B07_i28General_I_O.bOutput3 <-> API/Term 12 (PLC Output  )/Subterm 18 (Instrument Control )/Outputs/Instrument Control/User_Configurable_Output_3
//     PlcTask Outputs/GVL_IO.dw_B07_i28General_I_O.bOutput4 <-> API/Term 12 (PLC Output  )/Subterm 18 (Instrument Control )/Outputs/Instrument Control/User_Configurable_Output_4
//     PlcTask Outputs/GVL_IO.dw_B07_i28General_I_O.bOutput5 <-> API/Term 12 (PLC Output  )/Subterm 18 (Instrument Control )/Outputs/Instrument Control/User_Configurable_Output_5
//     PlcTask Outputs/GVL_IO.dw_B07_i28General_I_O.bOutput6 <-> API/Term 12 (PLC Output  )/Subterm 18 (Instrument Control )/Outputs/Instrument Control/User_Configurable_Output_6
//     PlcTask Outputs/GVL_IO.dw_B07_i28General_I_O.bOutput7 <-> API/Term 12 (PLC Output  )/Subterm 18 (Instrument Control )/Outputs/Instrument Control/User_Configurable_Output_7
//     PlcTask Outputs/GVL_IO.dw_B07_i28General_I_O.bOutput8 <-> API/Term 12 (PLC Output  )/Subterm 18 (Instrument Control )/Outputs/Instrument Control/User_Configurable_Output_8
//     PlcTask Outputs/GVL_IO.dw_B07_i28General_I_O.bOutput9 <-> API/Term 12 (PLC Output  )/Subterm 18 (Instrument Control )/Outputs/Instrument Control/User_Configurable_Output_9
//     PlcTask Outputs/GVL_IO.dw_B07_i28General_I_O.bReset <-> API/Term 12 (PLC Output  )/Subterm 18 (Instrument Control )/Outputs/Instrument Control/Reset
//     PlcTask Outputs/GVL_IO.dw_B07_i28General_I_O.bSetProgram[0] <-> API/Term 12 (PLC Output  )/Subterm 18 (Instrument Control )/Outputs/Desired Program Number[0]
//     PlcTask Outputs/GVL_IO.dw_B07_i28General_I_O.bSetProgram[1] <-> API/Term 12 (PLC Output  )/Subterm 18 (Instrument Control )/Outputs/Desired Program Number[1]
//     PlcTask Outputs/GVL_IO.dw_B07_i28General_I_O.bSetProgram[2] <-> API/Term 12 (PLC Output  )/Subterm 18 (Instrument Control )/Outputs/Desired Program Number[2]
//     PlcTask Outputs/GVL_IO.dw_B07_i28General_I_O.bSetProgram[3] <-> API/Term 12 (PLC Output  )/Subterm 18 (Instrument Control )/Outputs/Desired Program Number[3]
//     PlcTask Outputs/GVL_IO.dw_B07_i28General_I_O.bSetProgram[4] <-> API/Term 12 (PLC Output  )/Subterm 18 (Instrument Control )/Outputs/Desired Program Number[4]
//     PlcTask Outputs/GVL_IO.dw_B07_i28General_I_O.bSetProgram[5] <-> API/Term 12 (PLC Output  )/Subterm 18 (Instrument Control )/Outputs/Desired Program Number[5]
//     PlcTask Outputs/GVL_IO.dw_B07_i28General_I_O.bSetProgram[6] <-> API/Term 12 (PLC Output  )/Subterm 18 (Instrument Control )/Outputs/Desired Program Number[6]
//     PlcTask Outputs/GVL_IO.dw_B07_i28General_I_O.bSetProgram[7] <-> API/Term 12 (PLC Output  )/Subterm 18 (Instrument Control )/Outputs/Desired Program Number[7]
//     PlcTask Outputs/GVL_IO.dw_B07_i28General_I_O.bStart <-> API/Term 12 (PLC Output  )/Subterm 18 (Instrument Control )/Outputs/Instrument Control/Start
//     PlcTask Outputs/GVL_IO.dw_B07_i28General_I_O.bStop <-> API/Term 12 (PLC Output  )/Subterm 18 (Instrument Control )/Outputs/Instrument Control/Stop
//     PlcTask Outputs/GVL_IO.dw_B07_i28General_I_O.bVentHalt <-> API/Term 12 (PLC Output  )/Subterm 18 (Instrument Control )/Outputs/Instrument Control/Vent_Halt
//   LeakTesters/LeakTesters Instance <-> Device 2 (EL6631)/is2802
//     PlcTask Inputs/GVL_IO.dwBoxInfo[15].nPnIoBoxDiag <-> Inputs/PnIoBoxDiag
//     PlcTask Inputs/GVL_IO.dwBoxInfo[15].nPnIoBoxState <-> Inputs/PnIoBoxState
//     PlcTask Inputs/GVL_IO.dw_B06_IS2802M.aqsAcquisitionError <-> API/Term 3 (Acquisition Status)/Subterm 5 (Acquisition Status)/Inputs/Acquisition Status Register/Acquisition_Error
//     PlcTask Inputs/GVL_IO.dw_B06_IS2802M.aqsAcquisitionID <-> API/Term 3 (Acquisition Status)/Subterm 5 (Acquisition Status)/Inputs/Acquisition ID
//     PlcTask Inputs/GVL_IO.dw_B06_IS2802M.aqsExposureComplete <-> API/Term 3 (Acquisition Status)/Subterm 5 (Acquisition Status)/Inputs/Acquisition Status Register/Exposure_Complete
//     PlcTask Inputs/GVL_IO.dw_B06_IS2802M.aqsOnline <-> API/Term 3 (Acquisition Status)/Subterm 5 (Acquisition Status)/Inputs/Acquisition Status Register/Online
//     PlcTask Inputs/GVL_IO.dw_B06_IS2802M.aqsTriggerAcknowledge <-> API/Term 3 (Acquisition Status)/Subterm 5 (Acquisition Status)/Inputs/Acquisition Status Register/Acquisition_Trigger_Acknowledge
//     PlcTask Inputs/GVL_IO.dw_B06_IS2802M.aqsTriggerReady <-> API/Term 3 (Acquisition Status)/Subterm 5 (Acquisition Status)/Inputs/Acquisition Status Register/Acquisition_Trigger_Ready
//     PlcTask Inputs/GVL_IO.dw_B06_IS2802M.ccoCommandResultCode <-> API/Term 6 (Command Control)/Subterm 8 (Command Control)/Inputs/Command Result Code
//     PlcTask Inputs/GVL_IO.dw_B06_IS2802M.ccoCurrentJobID <-> API/Term 6 (Command Control)/Subterm 8 (Command Control)/Inputs/Current Job ID
//     PlcTask Inputs/GVL_IO.dw_B06_IS2802M.eesExternalEventStatus[0] <-> API/Term 7 (ExternalEvent Control)/Subterm 9 (ExternalEvent Control)/Inputs/ExternalEvent Status/Trigger_ExternalEvent_0_Acknowledge
//     PlcTask Inputs/GVL_IO.dw_B06_IS2802M.eesExternalEventStatus[1] <-> API/Term 7 (ExternalEvent Control)/Subterm 9 (ExternalEvent Control)/Inputs/ExternalEvent Status/Trigger_ExternalEvent_1_Acknowledge
//     PlcTask Inputs/GVL_IO.dw_B06_IS2802M.eesExternalEventStatus[2] <-> API/Term 7 (ExternalEvent Control)/Subterm 9 (ExternalEvent Control)/Inputs/ExternalEvent Status/Trigger_ExternalEvent_2_Acknowledge
//     PlcTask Inputs/GVL_IO.dw_B06_IS2802M.eesExternalEventStatus[3] <-> API/Term 7 (ExternalEvent Control)/Subterm 9 (ExternalEvent Control)/Inputs/ExternalEvent Status/Trigger_ExternalEvent_3_Acknowledge
//     PlcTask Inputs/GVL_IO.dw_B06_IS2802M.eesExternalEventStatus[4] <-> API/Term 7 (ExternalEvent Control)/Subterm 9 (ExternalEvent Control)/Inputs/ExternalEvent Status/Trigger_ExternalEvent_4_Acknowledge
//     PlcTask Inputs/GVL_IO.dw_B06_IS2802M.eesExternalEventStatus[5] <-> API/Term 7 (ExternalEvent Control)/Subterm 9 (ExternalEvent Control)/Inputs/ExternalEvent Status/Trigger_ExternalEvent_5_Acknowledge
//     PlcTask Inputs/GVL_IO.dw_B06_IS2802M.eesExternalEventStatus[6] <-> API/Term 7 (ExternalEvent Control)/Subterm 9 (ExternalEvent Control)/Inputs/ExternalEvent Status/Trigger_ExternalEvent_6_Acknowledge
//     PlcTask Inputs/GVL_IO.dw_B06_IS2802M.eesExternalEventStatus[7] <-> API/Term 7 (ExternalEvent Control)/Subterm 9 (ExternalEvent Control)/Inputs/ExternalEvent Status/Trigger_ExternalEvent_7_Acknowledge
//     PlcTask Inputs/GVL_IO.dw_B06_IS2802M.irInspectionID <-> API/Term 9 (Results - 64 bytes)/Subterm 11 (Results - 64 bytes)/Inputs/Inspection ID
//     PlcTask Inputs/GVL_IO.dw_B06_IS2802M.irInspectionResults <-> API/Term 9 (Results - 64 bytes)/Subterm 11 (Results - 64 bytes)/Inputs/Inspection Results
//     PlcTask Inputs/GVL_IO.dw_B06_IS2802M.irInspectionResultsCode <-> API/Term 9 (Results - 64 bytes)/Subterm 11 (Results - 64 bytes)/Inputs/Inspection Result Code
//     PlcTask Inputs/GVL_IO.dw_B06_IS2802M.isCommandCompleted <-> API/Term 5 (Inspection Status)/Subterm 7 (Inspection Status)/Inputs/Inspection Status Register/Command_Completed
//     PlcTask Inputs/GVL_IO.dw_B06_IS2802M.isCommandExecuting <-> API/Term 5 (Inspection Status)/Subterm 7 (Inspection Status)/Inputs/Inspection Status Register/Command_Executing
//     PlcTask Inputs/GVL_IO.dw_B06_IS2802M.isCommandFailed <-> API/Term 5 (Inspection Status)/Subterm 7 (Inspection Status)/Inputs/Inspection Status Register/Command_Failed
//     PlcTask Inputs/GVL_IO.dw_B06_IS2802M.isError <-> API/Term 5 (Inspection Status)/Subterm 7 (Inspection Status)/Inputs/Inspection Status Register/Error
//     PlcTask Inputs/GVL_IO.dw_B06_IS2802M.isErrorID <-> API/Term 5 (Inspection Status)/Subterm 7 (Inspection Status)/Inputs/Error ID
//     PlcTask Inputs/GVL_IO.dw_B06_IS2802M.isInspectionCompleted <-> API/Term 5 (Inspection Status)/Subterm 7 (Inspection Status)/Inputs/Inspection Status Register/Inspection_Completed
//     PlcTask Inputs/GVL_IO.dw_B06_IS2802M.isJobPassed <-> API/Term 5 (Inspection Status)/Subterm 7 (Inspection Status)/Inputs/Inspection Status Register/Job_Pass
//     PlcTask Inputs/GVL_IO.dw_B06_IS2802M.isResultsBufferOverrun <-> API/Term 5 (Inspection Status)/Subterm 7 (Inspection Status)/Inputs/Inspection Status Register/Results_Buffer_Overrun
//     PlcTask Inputs/GVL_IO.dw_B06_IS2802M.isResultsValid <-> API/Term 5 (Inspection Status)/Subterm 7 (Inspection Status)/Inputs/Inspection Status Register/Results_Valid
//     PlcTask Inputs/GVL_IO.dw_B06_IS2802M.isSetUserDataAcknowledge <-> API/Term 5 (Inspection Status)/Subterm 7 (Inspection Status)/Inputs/Inspection Status Register/User_Data_Set_Acknowledge
//     PlcTask Outputs/GVL_IO.dw_B06_IS2802M.aqcClearExposureComplete <-> API/Term 2 (Acquisition Control)/Subterm 4 (Acquisition Control)/Outputs/Acquisition Control Register/Clear_Exposure_Complete
//     PlcTask Outputs/GVL_IO.dw_B06_IS2802M.aqcSetOffline <-> API/Term 2 (Acquisition Control)/Subterm 4 (Acquisition Control)/Outputs/Acquisition Control Register/Set_In_Sight_Offline
//     PlcTask Outputs/GVL_IO.dw_B06_IS2802M.aqcTrigger <-> API/Term 2 (Acquisition Control)/Subterm 4 (Acquisition Control)/Outputs/Acquisition Control Register/Acquisition_Trigger
//     PlcTask Outputs/GVL_IO.dw_B06_IS2802M.aqcTriggerEnable <-> API/Term 2 (Acquisition Control)/Subterm 4 (Acquisition Control)/Outputs/Acquisition Control Register/Acquisition_Trigger_Enable
//     PlcTask Outputs/GVL_IO.dw_B06_IS2802M.cciCommandID <-> API/Term 6 (Command Control)/Subterm 8 (Command Control)/Outputs/Command ID
//     PlcTask Outputs/GVL_IO.dw_B06_IS2802M.eecExternalEventControl[0] <-> API/Term 7 (ExternalEvent Control)/Subterm 9 (ExternalEvent Control)/Outputs/ExternalEvent Control/Trigger_ExternalEvent_0
//     PlcTask Outputs/GVL_IO.dw_B06_IS2802M.eecExternalEventControl[1] <-> API/Term 7 (ExternalEvent Control)/Subterm 9 (ExternalEvent Control)/Outputs/ExternalEvent Control/Trigger_ExternalEvent_1
//     PlcTask Outputs/GVL_IO.dw_B06_IS2802M.eecExternalEventControl[2] <-> API/Term 7 (ExternalEvent Control)/Subterm 9 (ExternalEvent Control)/Outputs/ExternalEvent Control/Trigger_ExternalEvent_2
//     PlcTask Outputs/GVL_IO.dw_B06_IS2802M.eecExternalEventControl[3] <-> API/Term 7 (ExternalEvent Control)/Subterm 9 (ExternalEvent Control)/Outputs/ExternalEvent Control/Trigger_ExternalEvent_3
//     PlcTask Outputs/GVL_IO.dw_B06_IS2802M.eecExternalEventControl[4] <-> API/Term 7 (ExternalEvent Control)/Subterm 9 (ExternalEvent Control)/Outputs/ExternalEvent Control/Trigger_ExternalEvent_4
//     PlcTask Outputs/GVL_IO.dw_B06_IS2802M.eecExternalEventControl[5] <-> API/Term 7 (ExternalEvent Control)/Subterm 9 (ExternalEvent Control)/Outputs/ExternalEvent Control/Trigger_ExternalEvent_5
//     PlcTask Outputs/GVL_IO.dw_B06_IS2802M.eecExternalEventControl[6] <-> API/Term 7 (ExternalEvent Control)/Subterm 9 (ExternalEvent Control)/Outputs/ExternalEvent Control/Trigger_ExternalEvent_6
//     PlcTask Outputs/GVL_IO.dw_B06_IS2802M.eecExternalEventControl[7] <-> API/Term 7 (ExternalEvent Control)/Subterm 9 (ExternalEvent Control)/Outputs/ExternalEvent Control/Trigger_ExternalEvent_7
//     PlcTask Outputs/GVL_IO.dw_B06_IS2802M.icBufferResultsEnable <-> API/Term 4 (Inspection Control)/Subterm 6 (Inspection Control)/Outputs/Inspection Control Register/Enable_Results_Buffering
//     PlcTask Outputs/GVL_IO.dw_B06_IS2802M.icClearError <-> API/Term 4 (Inspection Control)/Subterm 6 (Inspection Control)/Outputs/Inspection Control Register/Clear_Error
//     PlcTask Outputs/GVL_IO.dw_B06_IS2802M.icExecuteCommand <-> API/Term 4 (Inspection Control)/Subterm 6 (Inspection Control)/Outputs/Inspection Control Register/Execute_Command
//     PlcTask Outputs/GVL_IO.dw_B06_IS2802M.icInspectionResultsAcknowledge <-> API/Term 4 (Inspection Control)/Subterm 6 (Inspection Control)/Outputs/Inspection Control Register/Acknowledge_Inspection_Results
//     PlcTask Outputs/GVL_IO.dw_B06_IS2802M.icSetUserData <-> API/Term 4 (Inspection Control)/Subterm 6 (Inspection Control)/Outputs/Inspection Control Register/Extended_User_Data_Set

// ---- DUTs/E_CameraJobChange.TcDUT
{attribute 'qualified_only'}
{attribute 'strict'}
TYPE E_CameraJobChange :
(
	WAITING_FOR_REQUEST := 50,
	LOAD_PROD_JOB := 200,
	LOAD_CALB_JOB := 300,
	GO_OFFLINE	  := 350,
	EXECUTE_COMMAND := 400,
	RESET_FLAG := 600
);
END_TYPE

// ---- DUTs/HeightMeasureFunction/E_HeighttMeasureProcess.TcDUT
{attribute 'qualified_only'}
{attribute 'strict'}
TYPE E_HeighttMeasureProcess :
(
	WAITING_ENABLE 					:= 0,
	WAITING_MEASURING_REQUEST		:= 20,
	CALIBRATIONBLOCK_METHOD			:= 40,
	GLODENPART_METHOD				:= 60,
	WAITING_FOR_MEASURE				:= 80,
	RESET							:= 100,
	SENSOR_STUCK_EVALUATION			:= 120,
	Manual_Mode						:= 140
	
);
END_TYPE

// ---- DUTs/IO/st_IS2802M.TcDUT
TYPE st_IS2802M :
STRUCT
	
// Camera Output 
    aqcTriggerEnable               AT%Q*       : BOOL;
    aqcTrigger                     AT%Q*       : BOOL;
    aqcClearExposureComplete       AT%Q*       : BOOL;
    aqcSetOffline                  AT%Q*       : BOOL;
	eecExternalEventControl        AT%Q*       : ARRAY[0..7] OF BOOL;
    icBufferResultsEnable          AT%Q*       : BOOL;
    icInspectionResultsAcknowledge AT%Q*       : BOOL;
    icSetUserData                  AT%Q*       : BOOL;
    icExecuteCommand               AT%Q*       : BOOL;
    icClearError                   AT%Q*       : BOOL;
	cciCommandID                   AT%Q*       : UINT;
// Camera Input	
    aqsTriggerReady                AT%I*       : BOOL; 
    aqsTriggerAcknowledge          AT%I*       : BOOL; 
    aqsExposureComplete            AT%I*       : BOOL; 
    aqsAcquisitionError            AT%I*       : BOOL; 
    aqsOfflineReason               AT%I*       : BOOL; 
    aqsOnline                      AT%I*       : BOOL; 
    aqsAcquisitionID               AT%I*       : UINT; 
    ccoCurrentJobID                AT%I*       : UINT;
    ccoCommandResultCode           AT%I*       : UINT;		
	eesExternalEventStatus         AT%I*       : ARRAY[0..7] OF BOOL;
    isInspectionCompleted          AT%I*       : BOOL; 
    isResultsBufferOverrun         AT%I*       : BOOL; 
    isResultsValid                 AT%I*       : BOOL; 
    isCommandExecuting             AT%I*       : BOOL; 
    isCommandCompleted             AT%I*       : BOOL; 
    isCommandFailed                AT%I*       : BOOL; 
    isSetUserDataAcknowledge       AT%I*       : BOOL; 
    isJobPassed                    AT%I*       : BOOL; 
    isError                        AT%I*       : BOOL; 
    isErrorID                      AT%I*       : UINT; 
	irInspectionID                 AT%I*       : UINT; 
    irInspectionResultsCode        AT%I*       : UINT; 
    irInspectionResults            AT%I*       : ARRAY[0..63]OF BYTE; 
	
	
END_STRUCT
END_TYPE

// ---- DUTs/IO/ST_DL_PN1.TcDUT
TYPE ST_DL_PN1 :
STRUCT
// Terminal 	
dldCurrValProp   AT %I*  :BOOL;
dldWarningStat   AT %I*  :BOOL;
dldErrorStt      AT %I*  :BOOL;
dldExtInpResp    AT %I*  :ARRAY[1..5] OF BOOL;
dldExtInpRespOut AT %Q*  :ARRAY[1..5] OF BOOL;
//GT2 Keyence Sensor 1
gt2_1_1Output       AT %I*  :ARRAY[1..5] OF BOOL;
gt2_1_1CurrValInv   AT %I*  :BOOL;
gt2_1_1CurrValUndR  AT %I*  :BOOL;
gt2_1_1CurrValOvrR  AT %I*  :BOOL;
gt2_1_1WarningStat  AT %I*  :BOOL;
gt2_1_1ErrorStat    AT %I*  :BOOL;
gt2_1_1ExtInpRes    AT %I*  :ARRAY[1..5] OF BOOL;
gt2_1_1CurrentValue AT %I*  :DINT;
gt2_1_1ExtInpResOut AT %Q*  :ARRAY[1..5] OF BOOL;
//GT2 Keyence Sensor 2	
gt2_1_2Output       AT %I*  :ARRAY[1..5] OF BOOL;
gt2_1_2CurrValInv   AT %I*  :BOOL;
gt2_1_2CurrValUndR  AT %I*  :BOOL;
gt2_1_2CurrValOvrR  AT %I*  :BOOL;
gt2_1_2WarningStat  AT %I*  :BOOL;
gt2_1_2ErrorStat    AT %I*  :BOOL;
gt2_1_2ExtInpRes    AT %I*  :ARRAY[1..5] OF BOOL;
gt2_1_2CurrentValue AT %I*  :DINT;
gt2_1_2ExtInpResOut AT %Q*  :ARRAY[1..5] OF BOOL;
//GT2 Keyence Sensor 3
gt2_1_3Output       AT %I*  :ARRAY[1..5] OF BOOL;
gt2_1_3CurrValInv   AT %I*  :BOOL;
gt2_1_3CurrValUndR  AT %I*  :BOOL;
gt2_1_3CurrValOvrR  AT %I*  :BOOL;
gt2_1_3WarningStat  AT %I*  :BOOL;
gt2_1_3ErrorStat    AT %I*  :BOOL;
gt2_1_3ExtInpRes    AT %I*  :ARRAY[1..5] OF BOOL;
gt2_1_3CurrentValue AT %I*  :DINT;
gt2_1_3ExtInpResOut AT %Q*  :ARRAY[1..5] OF BOOL;
//GT2 Keyence Sensor 4
gt2_2Output       AT %I*  :ARRAY[1..5] OF BOOL;
gt2_2CurrValInv   AT %I*  :BOOL;
gt2_2CurrValUndR  AT %I*  :BOOL;
gt2_2CurrValOvrR  AT %I*  :BOOL;
gt2_2WarningStat  AT %I*  :BOOL;
gt2_2ErrorStat    AT %I*  :BOOL;
gt2_2ExtInpRes    AT %I*  :ARRAY[1..5] OF BOOL;
gt2_2CurrentValue AT %I*  :DINT;
gt2_2ExtInpResOut AT %Q*  :ARRAY[1..5] OF BOOL;
END_STRUCT
END_TYPE

// ---- DUTs/ST_HeightLimits.TcDUT
TYPE ST_HeightLimits :
STRUCT
	
	nHigh					: REAL;
	nLow					: REAL;

END_STRUCT
END_TYPE

// ---- DUTs/ST_HeightMeasurement2.TcDUT
TYPE ST_HeightMeasurement2 :
STRUCT
	//INPUTS
	aSensorCurrentValue							: ARRAY[1..4] OF REAL;		
	bEnable										: BOOL;
	bMeasurementRequest							: BOOL;
	aTolerance									: ARRAY[1..3] OF REAL;
	bAcknowledge								: BOOL;
	nDistanceBetweenPoints						: ARRAY[1..3] OF REAL;
	anDistanceSetPoint							: ARRAY[1..3] OF REAL;
	EHeighttMeasureProcess						: E_HeighttMeasureProcess;
	//OUTPUTS
	bBusy										: BOOL;
	bComplete									: BOOL;
	bEnableo									: BOOL;
	aPass										: ARRAY[1..5] OF BOOL; //5 Final Result
	aFail										: ARRAY[1..5] OF BOOL; //5 Final Result
	aMinLimitCalibrationBlock					: ARRAY[1..3] OF REAL;
	aMaxLimitCalibrationBlock					: ARRAY[1..3] OF REAL;
	aDistanceBetweenProbes						: ARRAY[1..3] OF REAL; //1 Probe 1 to probe zero
	abSensorStuck								: ARRAY[1..4] OF BOOL;
	nFixedPoint									: ARRAY[1..4] OF REAL;
	aScaledSensorCurrentValue					: ARRAY[1..4] OF REAL;
	
	
END_STRUCT
END_TYPE

// ---- DUTs/ST_Nest.TcDUT
TYPE ST_Nest :
STRUCT
		 

	 
     bNestPartProced    : BOOL;
     bNestPartOK        : BOOL;
	 bNestPresent       : BOOL;

	 
	 bHeightPass		: BOOL;
	 bVisionPass		: BOOL;
	 bLeakPass			: BOOL;
	 bPiecePass			: BOOL;
	 
	 bHeightReject		: BOOL;
	 bVisionReject		: BOOL;
	 bLeakReject		: BOOL;	
	 bPieceReject		: BOOL; 
	 
	 sHeightHMI			: WSTRING;
	 sVisionHMI			: WSTRING;
	 sLeakHMI			: WSTRING;
	 sPieceHMI			: WSTRING;

	 nDistance			: ARRAY[1..3] OF REAL;
	 nTarget			: ARRAY[1..3] OF REAL;	

 
	 sDate				: STRING;
	 sTime				: STRING;

END_STRUCT
END_TYPE

// ---- DUTs/ST_PartsInspection.TcDUT
TYPE ST_PartsInspection :
STRUCT
	
	nVisionPartsGood				: DINT;
	nVisionTotalPartsGood			: DINT;
	nVisionPartsFailed				: DINT;
	nVisionTotalPartsFailed			: DINT;
	
	nHeightPartsGood				: DINT;
	nHeightTotalPartsGood			: DINT;
	nHeightPartsFailed				: DINT;
	nHeightTotalPartsFailed			: DINT;
	
	nHeightDistancePartsGood		: ARRAY[1..4] OF DINT;
	nHeightDistanceTotalPartsGood	: ARRAY[1..4] OF DINT;
	nHeightDistancePartsFailed		: ARRAY[1..4] OF DINT;
	nHeightDistanceTotalPartsFailed	: ARRAY[1..4] OF DINT;
	
	nLeakPartsGood					: DINT;
	nLeakTotalPartsGood				: DINT;
	nLeakPartsFailed				: DINT;
	nLeakTotalPartsFailed			: DINT;
	
	nPartsGood						: DINT;
	nTotalPartsGood					: DINT;
	nPartsFailed					: DINT;
	nTotalPartsFailed				: DINT;					
	
	bPartok							: BOOL;
	bPartFail						: BOOL;
END_STRUCT
END_TYPE

// ---- GVLs/GVL_HMI_GLOBAL.TcGVL
{attribute 'qualified_only'}
VAR_GLOBAL
	
	//User Log, Shut down, Quit HMI
	bQuitHmi						: BOOL;
	sUserGroup						: STRING;
	sUserGroup2						: STRING;
	sUserName						: STRING;
	bLogOut							: BOOL;
	bUserLogedIntSignal				: BOOL;
	bShutDown						: BOOL;
	
	
	
	
	
	//General
	bStopButton						: BOOL;
	bStartButton					: BOOL;
	bResetButton					: BOOL;
	nRegionMain						: INT;
	bTrigerCamMan					: BOOL;
	bResetGoodParts					: BOOL;
	bResetFailedParts				: BOOL;
	
	aEventTexts						: ARRAY [0..767] OF T_MaxSTring; //Event texts - set only once
	bEventTextsSet					: BOOL;
	aEventFlags						: ARRAY [0..767] OF BOOL;		//All event states combined from master na stations
	aActiveEvents					: ARRAY [0..39] OF T_MaxSTring;	//Active events - connected to Alarm scree in HMI	
	stActiveEventsHMI				: ARRAY [0..39] OF ST_ActiveEventsHMI;
	
	sMessageToOperator				: WSTRING(200);
	sActualProcess					: WSTRING(200);
	aIOScreen						: ARRAY [0..10] OF STRING(200);
	aManualScreen					: ARRAY [0..2] OF STRING(200);
	bResetPassAndFail				: BOOL;
	bEnableManualMode				: BOOL;
	bRejectPieceAcknowledge			: BOOL;
	bRejectPieceDialogTrig			: BOOL;
	bAutocycleFaultDialog			: BOOL;
	
	
	
	// ------ Screen Info / Data -----------	
	sSystemDate					: STRING;
	sSystemTime					: STRING;
	ntAMSNetID					: T_AmsNetId := '172.18.237.82.1.1';
	
	
	
	//Camera
	bManualModeOff					: ARRAY[1..2] OF BOOL;
	bResetCamMan					: BOOL;
	sInfoCamMan						: STRING;
	bLoadProductionJob				: BOOL;
	bLoadCalibrationJob				: BOOL;
	bEnableTrigerMan				: BOOL;
	bVisionPass						: BOOL;
	bResetVisionGoodParts			: BOOL;
	bResetVisionBadParts			: BOOL;
	
	
	//Leak Tester
	bLeakTestPass					: BOOL;
	uSetLeakProgramID				: USINT;
	bSetLeakProgramID				: BOOL;
	bResetLeakMan					: BOOL;
	bStartLeakMan					: BOOL;
	bStopLeakMan					: BOOL;
	bLoadLeakProg					: BOOL;
	uNewLeakProgID					: USINT;
	
	
	
	bResetLeakGoodParts				: BOOL;
	bResetLeakBadParts				: BOOL;
	
	
	
	
	//Height Tester
	bHeightTestPass					: BOOL;
	bResetHeightGoodParts			: BOOL;
	bResetHeightFailParts			: BOOL;
	bManualHeightTrigger			: BOOL;
	aResetHeightSensorGoodParts		: ARRAY[1..4] OF BOOL;
	aResetHeightSensorBadParts		: ARRAY[1..4] OF BOOL;
	
	
	bSetSetPointsHeightTest			: BOOL;
	bManualMeasureHeightTest		: BOOL;
	aGeneralPassHeightTest			: ARRAY[1..5] OF BOOL;
	aGeneralFailHeightTest			: ARRAY[1..5] OF BOOL;
	
	anValueScaledHeightTest			: ARRAY[1..4] OF DINT;
	
	aSensorSetPointsHeightTest		: ARRAY[1..4] OF DINT;
	
	nHeightMeasureStateValue		: ARRAY[1..4] OF DINT;
	bProbesPositionOk				: BOOL;
	

	

	
	

END_VAR
VAR_GLOBAL PERSISTENT
	
	aStatistics					: ARRAY [1..201] OF ST_Nest;//LA** 04092025 >> : ARRAY [1..200] OF ST_Nest;
	stAlarmHistory				:ARRAY [00..250] OF ST_AlarmHistory;
	aEventLog					:ARRAY [0..250] OF T_MaxSTring;	//Event log - connected to alarm history in HMI	
	aTimeLog					:ARRAY [0..250] OF T_MaxSTring;
	aDateLog					:ARRAY [0..250] OF T_MaxSTring;
	aMinLimitHeightTest				: ARRAY[1..4] OF DINT;
	aMaxLimitHeightTest				: ARRAY[1..4] OF DINT;	
		
END_VAR

// ---- GVLs/GVL_IO.TcGVL
{attribute 'qualified_only'}
VAR_GLOBAL
	
    //--------------------------------------------------------------------------------------------------------

    dwTerminalInfo                                          : ARRAY[0..20] OF  st_Terminal_Info; // all terminal's status information 
	dwBoxInfo                                               : ARRAY[15..17] OF st_Box_Info;//Camera, Leak, Height
	//--------------------------------------------------------------------------------------------------------
	
	(* Terminal *)
	
	//	dw_T01_EK1100                                                	| EtherCAT Coupler 
	//	dw_T02_EL6070-0033                                           	| EtherCAT Terminal, license key for TwinCAT 3.1
	
	dw_T02_EL1809                                                		: st_EL1809; //16 Channel Digital Input ( 24VDC ) 
	dw_T03_EL2809                                                		: st_EL2809; // 16 Channel Digital Output ( 24VDC )
	//dw_T04_EL6631                                                	| EtherCAT Terminal, 2-port communication interface, PROFINET RT, controller - Data for Box's MDU1020 and SR2000W
 	//  dw_T05_EL9011                                                	| Bus end cover for E-bus contacts
	dw_B06_IS2802M                                               		: st_IS2802M;
	
	dw_B07_i28General_I_O												: st_i28General_I_O;
	dw_B07_i28LastResult												: st_i28LasResult;
	dw_B07_i28LiveMeasurement											: st_i28LiveMeasurement;
	
	dw_B08_DL_PN1                                                		: ST_DL_PN1; // Keyence GT2 Position Sensors 
	
	
END_VAR

// ---- GVLs/GVL_MASTER.TcGVL
{attribute 'qualified_only'}
VAR_GLOBAL
	(*-----------------------------------------------------------------------------------------------------------------*)
	// System Pulses 
	bFlash1Hz						: BOOL;
	bFlash2Hz						: BOOL;
	bFlash4Hz				   		: BOOL;
	bFlash10Hz						: BOOL;
	bFlash10BHz        		  		: BOOL;
	bFlash100Hz      	      		: BOOL;
	bFlashScale       	      		: BOOL;
	bFlashScale4       		  		: BOOL;
	bFlashScale5        	  		: BOOL;
	bFlashingFreq2			  		: BOOL;
	bFlashScaleFast       	  		: BOOL;
	
//Master Control
	stMachineStatus					: ST_MachineStatusStruct;	
	stMasterControl					: ST_MasterControlStruct;
  	stStationSruct                  : ARRAY[0..5] OF ST_StandardStationStruct; (* Station 0 - Master
                                                                                  Station 1 - Height test 
	                                                                              Station 2 - Leak test
																				  Station 3 - Vision test 
                                                                                   *)
	bHeightTestacknowledge			: BOOL;
	
																				   
	stNest							: ST_Nest;                                                                        
	stAlarms                        : ARRAY [0..3] OF ST_Events;
	
	bManualModeTrigger				: BOOL;
	abSensorStuck					: ARRAY[1..4] OF BOOL;
	anValueBeforeMeasurement		: ARRAY[1..4] OF DINT;
	aSensorCurrentValue				: ARRAY[1..4] OF DINT;
	
																				   

END_VAR

// ---- GVLs/GVL_PERSIST.TcGVL
{attribute 'qualified_only'}
VAR_GLOBAL PERSISTENT
	
stPartsInspection			: ST_PartsInspection;
stUserLogHMI				: ARRAY[0..250] OF ST_UserLogHMI;
UserId						: UINT;
ast_i28LasResult            : ARRAY [0..250] OF st_i28LasResult;
nLeakTestID					: UINT;

nCycleNumber				: INT;

aSensorSetPointsHeightTest		: ARRAY[1..4] OF DINT;
aTolerancesHeightTest			: ARRAY[1..4] OF DINT;

stHeightLimits					: ST_HeightLimits;





	
	
END_VAR

// ---- POUs/A_Master/Main_Master.TcPOU
PROGRAM Main_Master
VAR
	i                       :INT; //Int to handle user log index	
	k						:INT; //Int to handle user log index
	j						:INT;
	l						:INT;
	
	//////UserLog
	
	sUserGroupID			:	STRING;
	nSize					:	UDINT					:=9;
	nLen					:	UDINT					:=18;
	npos					:	UDINT					:=1;
	tonUserLogOut           :	Tc2_Standard.TON;
	fbStringFormatter       :	Tc2_Utilities.FB_FormatString;
	fbEventLogger			:	FB_EventLog;
	rUserLoggedIn			: 	R_TRIG;
	tUserLoggedIn			: 	TON;
	bFirstScan				:   BOOL;
	tFirstScan				:   TON;

	bUserLoggedIn			: 	BOOL;
	

	
	
	/////ShutDown&Quit
	closeChrome 			: 	NT_StartProcess;	
	ntShutdown					: TC2_Utilities.NT_Shutdown;
	ntError						: BOOL;
	ntBusy						: BOOL;
	ntErrorID					: UDINT;

	
	
	/////General

END_VAR

PRG_FaultHandling(aAlarms := GVL_Master.stAlarms );
PRG_Fault_HeightTest(aAlarms := GVL_Master.stAlarms);
PRG_Fault_LeakTest(aAlarms := GVL_Master.stAlarms);
PRG_Fault_VisionTest(aAlarms := GVL_Master.stAlarms);

PRG_MachineStatus();
PRG_MasterCycle(stStationStruct:= GVL_Master.stStationSruct[0]);
PRG_MasterSystemTime();
ACT_ShutdownAndQuit();
ACT_UserLog();
MapUnitEventsToHmi();
PRG_HMI();
PRG_Puls();
ACT_FirstScan();
PRG_TerminBoxInfo();

//gfggf




PRG_LeakTestEvents_Info();





//Stations
PRG_HeightTest(stStationStruct:= GVL_Master.stStationSruct[1]);
PRG_LeakTest(stStationStruct:= GVL_Master.stStationSruct[2]);
PRG_VisionTest(stStationStruct:= GVL_Master.stStationSruct[3]);



fbEventLogger(	bEnable       	:= PRG_MasterSystemTime.bReadyToRead AND GVL_MASTER.stMasterControl.bPowerUpTimerComplete,
			    sDateTime     	:= PRG_MasterSystemTime.sDateTimeSpaces,
			    aEventFlags   	:= GVL_HMI_GLOBAL.aEventFlags,
			    aEventTexts   	:= GVL_HMI_GLOBAL.aEventTexts,
			    aActiveEvents 	:= GVL_HMI_GLOBAL.aActiveEvents,
			    aEventLog     	:= GVL_HMI_GLOBAL.aEventLog,
				siDate			:= GVL_HMI_GLOBAL.sSystemDate,
				siTime			:= GVL_HMI_GLOBAL.sSystemTime,
				soDate			:= GVL_HMI_GLOBAL.aDateLog,
				soTime			:= GVL_HMI_GLOBAL.aTimeLog
);



 

IF GVL_MASTER.bFlashScale THEN
FOR j := 0 TO 39 DO
	
GVL_HMI_GLOBAL.stActiveEventsHMI[j].sActiveEvents := GVL_HMI_GLOBAL.aActiveEvents[j];
END_FOR
FOR l:=0 TO 250 DO
	
	GVL_HMI_GLOBAL.stAlarmHistory[l].sEventlog 	:= GVL_HMI_GLOBAL.aEventLog[l];
	GVL_HMI_GLOBAL.stAlarmHistory[l].sDate		:= GVL_HMI_GLOBAL.aDateLog[l];
	GVL_HMI_GLOBAL.stAlarmHistory[l].sTime		:= GVL_HMI_GLOBAL.aTimeLog[l];
END_FOR
ELSE 
	
j:=0; 
l:=0;

END_IF

ACTION ACT_FirstScan:
tFirstScan(IN := NOT bFirstScan, PT := T#5S);
END_ACTION

ACTION ACT_ShutdownAndQuit:
closeChrome(
    NetId := '',
    PathStr := 'C:\Windows\System32\mshta vbscript:Execute("CreateObject(""WScript.Shell"").Run ""powershell -c',
    DirName := 'C:\Windows\System32\WindowsPowerShell\v1.0',
    ComndLine := 'taskkill /F /IM chrome.exe /T"", 0: window.close")',
    Start := GVL_HMI_GLOBAL.bQuitHmi,
    TmOut := DEFAULT_ADS_TIMEOUT
);
 
GVL_HMI_GLOBAL.bQuitHmi:= FALSE;

ntShutdown(NETID := GVL_HMI_GLOBAL.ntAMSNetID, DELAY := 5, START := GVL_HMI_GLOBAL.bShutDown, BUSY => ntBusy, ERR => ntError, ERRID => ntErrorID);
END_ACTION

ACTION ACT_UserLog:

//Getting user group

Tc2_Utilities.DELETE2( ADR(GVL_HMI_GLOBAL.sUserGroup), ADR(sUserGroupID), NSize, Nlen, nPos) ;

IF sUserGroupID = 'Administ' THEN
	
	GVL_HMI_GLOBAL.sUserGroup2 := 'Administrator';

ELSE GVL_HMI_GLOBAL.sUserGroup2 := sUserGroupID;
	

END_IF


//Logout 

tonUserLogOut( IN := (sUserGroupID = 'Administ' OR sUserGroupID ='Engineer') AND GVL_HMI_GLOBAL.bUserLogedIntSignal , PT := T#10M);

IF tonUserLogOut.Q AND (sUserGroupID = 'Administ' OR sUserGroupID ='Engineer') THEN
	
	GVL_HMI_GLOBAL.bLogOut 	:= TRUE;

	ELSE GVL_HMI_GLOBAL.bLogOut := FALSE;

END_IF

tUserLoggedIn( IN := GVL_HMI_GLOBAL.bUserLogedIntSignal, PT := T#2S);

rUserLoggedIn( CLK := tUserLoggedIn.Q);


IF rUserLoggedIn.Q THEN
	
	FOR i :=200 TO 1 BY (-1) DO
		GVL_PERSIST.stUserLogHMI[i]	:= GVL_PERSIST.stUserLogHMI[i-1];
	END_FOR
	
	GVL_PERSIST.stUserLogHMI[0].UserLog := GVL_HMI_GLOBAL.sUserName;
	GVL_PERSIST.stUserLogHMI[0].UserLogTime := GVL_HMI_GLOBAL.sSystemTime;
	GVL_PERSIST.stUserLogHMI[0].UserLogDate := GVL_HMI_GLOBAL.sSystemDate;

END_IF
END_ACTION

METHOD MapUnitEventsToHMI : BOOL
VAR_INPUT
END_VAR

VAR
	i		:INT; 	//Unit index
	j		:INT;	//Unit event index
	k		:INT; 	//HMI event index	
END_VAR
//Set event texts first
IF GVL_Master.stAlarms[0].bEventTextsSet AND
   GVL_Master.stAlarms[1].bEventTextsSet AND
   GVL_Master.stAlarms[2].bEventTextsSet AND
   GVL_Master.stAlarms[3].bEventTextsSet AND
   NOT GVL_HMI_GLOBAL.bEventTextsSet 
THEN
	SetEventTexts();
		
	GVL_HMI_GLOBAL.bEventTextsSet := TRUE;
END_IF

//Map events from master and stations into HMI events
IF GVL_HMI_GLOBAL.bEventTextsSet THEN
	k := 0; 
	FOR i := 0 TO 3 DO
		FOR j := 0 TO 128 - 1 DO
			GVL_HMI_GLOBAL.aEventFlags[k] := GVL_Master.stAlarms[i].aEventFlags[j];
			k := k + 1;
		END_FOR
	END_FOR
END_IF
END_METHOD

METHOD SetEventTexts : BOOL
VAR_INPUT
END_VAR
VAR
	i				:INT; 	//Unit index
	j				:INT;	//HMI event index
	k				:INT;	//
END_VAR
//Set global event texts based on unit event texts (master and stations
k := 0;
FOR i := 0 TO 3 DO
	//For each unit (master, station1, station2)
	//Alarm texts
	FOR j := 0 TO 99 DO
		fbStringFormatter(	sFormat := 'Alarm No. %d - %s', 
					 	arg1 := F_INT(k), 
						arg2 := F_String(GVL_Master.stAlarms[i].aEventTexts[j]),
						sOut => GVL_HMI_GLOBAL.aEventTexts[k]);
						
		k := k + 1; //Increment global events index
	END_FOR
	
	//Messages
	FOR j := 100 TO 127 DO
		fbStringFormatter(	sFormat := 'Message No. %d - %s', 
					 		arg1 := F_INT(k), 
							arg2 := F_String(GVL_Master.stAlarms[i].aEventTexts[j]),
							sOut => GVL_HMI_GLOBAL.aEventTexts[k]);
							
		k := k + 1; //Increment global events index
	END_FOR
END_FOR
END_METHOD

END_PROGRAM

// ---- POUs/A_Master/PRG_FaultHandling.TcPOU
PROGRAM PRG_FaultHandling
VAR
	
	i							: INT;
	bFlagResetOn				: BOOL;
	bStationCycleFaultFlag		: BOOL;




END_VAR
VAR_IN_OUT

  aAlarms  : ARRAY[0..3] OF ST_Events;
END_VAR

ACT_FaultTrig();

(************************************** Faults reset **********************************************)
IF   GVL_HMI_GLOBAL.bResetButton THEN 
	FOR i := 0 TO 127 DO
		GVL_MASTER.stAlarms[0].aEventFlags[i] := FALSE;
	END_FOR
END_IF


//===============================================================
//Initialize event texts on first scan
IF NOT GVL_MASTER.stAlarms[0].bEventTextsSet THEN
	SetEventTexts();
	GVL_MASTER.stAlarms[0].bEventTextsSet := TRUE;
END_IF
IF NOT GVL_MASTER.stAlarms[0].bEventTextsSet THEN
	GVL_MASTER.stAlarms[0].bEventTextsSet := FALSE;
END_IF


(***************************************************************************************************)
//Immediate fault
GVL_MASTER.stAlarms[0].bImmediateFault := FALSE;
FOR i := 0 TO 32DO
	GVL_MASTER.stAlarms[0].bImmediateFault := GVL_MASTER.stAlarms[0].bImmediateFault OR GVL_MASTER.stAlarms[0].aEventFlags[i];
END_FOR

//Cycle stop fault
GVL_MASTER.stAlarms[0].bCycleStopFault := FALSE;
FOR i := 33 TO 79 DO
	GVL_MASTER.stAlarms[0].bCycleStopFault := GVL_MASTER.stAlarms[0].bCycleStopFault OR GVL_MASTER.stAlarms[0].aEventFlags[i];
END_FOR

//Cycle stop request
GVL_MASTER.stAlarms[0].bCycleStopRequest := FALSE;
FOR i := 80 TO 99 DO
	GVL_MASTER.stAlarms[0].bCycleStopRequest := GVL_MASTER.stAlarms[0].bCycleStopRequest OR GVL_MASTER.stAlarms[0].aEventFlags[i];
END_FOR


(**************************** Master Fault Monitors ***********************************************)
(* Station Immediate Fault Monitor *)
GVL_MASTER.stMasterControl.bNoStationImmediateFault := 	NOT GVL_MASTER.stAlarms[0].bImmediateFault AND NOT GVL_MASTER.stAlarms[1].bImmediateFault AND
                                            			NOT GVL_MASTER.stAlarms[2].bImmediateFault AND NOT GVL_MASTER.stAlarms[3].bImmediateFault;

(**************************************************************************************************)
(**************************** Cycle stop falt  **************************************)
bStationCycleFaultFlag := NOT GVL_MASTER.stAlarms[0].bCycleStopFault AND NOT GVL_MASTER.stAlarms[1].bCycleStopFault AND
                          NOT GVL_MASTER.stAlarms[2].bCycleStopFault AND NOT GVL_MASTER.stAlarms[3].bCycleStopFault;

(**************************** Master Immediate Fault Monitor **************************************)
GVL_MASTER.stMasterControl.bNoMachineImmediateFault := NOT GVL_MASTER.stAlarms[0].bImmediateFault AND NOT GVL_MASTER.stAlarms[1].bImmediateFault AND
                                            NOT GVL_MASTER.stAlarms[2].bImmediateFault AND NOT GVL_MASTER.stAlarms[3].bImmediateFault;

									
(**************************************************************************************************)

(* Master Cycle Stop Fault Monitor *)
GVL_MASTER.stMasterControl.bNoCycleStopFault := NOT GVL_MASTER.stAlarms[0].bCycleStopFault AND NOT GVL_MASTER.stAlarms[1].bCycleStopFault
												AND NOT GVL_MASTER.stAlarms[2].bCycleStopFault AND NOT GVL_MASTER.stAlarms[3].bCycleStopFault;

ACTION ACT_FaultTrig:
(**************************************************************************************************)
(**************************** Master Immediate Fault Stop *****************************************)
(**************************************************************************************************)

//Beckhoff EL1809 Not Operational
IF NOT GVL_MASTER.stMachineStatus.bSystemPowerUp AND GVL_IO.dwTerminalInfo[3].nTerminal_State<>8 THEN
	GVL_MASTER.stAlarms[0].aEventFlags[33] := TRUE;
END_IF
//Beckhoff EL2809 Not Operational
IF NOT GVL_MASTER.stMachineStatus.bSystemPowerUp AND GVL_IO.dwTerminalInfo[4].nTerminal_State<>8 THEN
	GVL_MASTER.stAlarms[0].aEventFlags[34] := TRUE;
END_IF
//Cognex  IS2801M Connection Erro
IF NOT GVL_MASTER.stMachineStatus.bSystemPowerUp AND GVL_IO.dwBoxInfo[15].nPnIoBoxState<>0 THEN
	GVL_MASTER.stAlarms[0].aEventFlags[35] := TRUE;
END_IF
//External Error - Cognex Camera ERROR
IF GVL_IO.dw_B06_IS2802M.isError   THEN // 
	GVL_MASTER.stAlarms[0].aEventFlags[36] := TRUE;
END_IF
//Cognex  IS2801M Diagnostic Error
IF NOT GVL_MASTER.stMachineStatus.bSystemPowerUp AND GVL_IO.dwBoxInfo[15].nPnIoBoxDiag=1 THEN
	GVL_MASTER.stAlarms[0].aEventFlags[37] := TRUE;
END_IF
//System stopping timeout
GVL_MASTER.stAlarms[0].aEventTimers[38](IN := ( GVL_MASTER.stMachineStatus.bSystemStopping ), PT := T#20S);
IF GVL_MASTER.stAlarms[0].aEventTimers[38].Q THEN
	GVL_MASTER.stAlarms[0].aEventFlags[38] := TRUE;	
END_IF
//User not Log In
GVL_MASTER.stAlarms[0].aEventTimers[39](IN := (NOT GVL_HMI_GLOBAL.bUserLogedIntSignal), PT := T#40MS);
IF GVL_MASTER.stAlarms[0].aEventTimers[39].Q THEN
	GVL_MASTER.stAlarms[0].aEventFlags[39] := TRUE;	
END_IF
//User LOG-Off Timeout Manual Mode
GVL_MASTER.stAlarms[0].aEventTimers[40](IN:= ((NOT GVL_HMI_GLOBAL.bUserLogedIntSignal) AND GVL_MASTER.stMachineStatus.bManualMode),PT:= T#1S); 
IF GVL_MASTER.stAlarms[0].aEventTimers[40].Q THEN
	GVL_MASTER.stAlarms[0].aEventFlags[40] := TRUE;
END_IF
//Keyence DL-P1 Error
IF GVL_IO.dw_B08_DL_PN1.dldErrorStt THEN
	GVL_MASTER.stAlarms[0].aEventFlags[41] := TRUE;
END_IF
//10 Min Auto cycle stop
IF PRG_MasterCycle.bAutoCycleStop  THEN //
	GVL_MASTER.stAlarms[0].aEventFlags[80] := TRUE;
END_IF
//Autocyle Timeout 
GVL_MASTER.stAlarms[0].aEventTimers[42](IN:= GVL_MASTER.stStationSruct[0].bStationInProgress, PT :=T#10M ); 
IF GVL_MASTER.stAlarms[0].aEventTimers[42].Q THEN
	GVL_MASTER.stAlarms[0].aEventFlags[42] := TRUE;
END_IF
//Part removed during process
IF GVL_Master.stStationSruct[0].nState > 1000 AND GVL_Master.stStationSruct[0].nState < 2000 AND NOT GVL_IO.dw_T02_EL1809.iPartPresent THEN
	GVL_MASTER.stAlarms[0].aEventFlags[43] := TRUE;
END_IF
//Clamp toggled before requested
IF GVL_Master.stStationSruct[0].nState > 1000 AND GVL_Master.stStationSruct[0].nState <= 1136 AND GVL_IO.dw_T02_EL1809.iCalmpClosed THEN
	GVL_MASTER.stAlarms[0].aEventFlags[44] := TRUE;
END_IF
//Clamp toggled before requested
IF GVL_Master.stStationSruct[0].nState > 1142 AND GVL_Master.stStationSruct[0].nState < 1700 AND NOT GVL_IO.dw_T02_EL1809.iCalmpClosed THEN
	GVL_MASTER.stAlarms[0].aEventFlags[45] := TRUE;
END_IF
//Press Acknowledge
IF GVL_HMI_GLOBAL.bAutocycleFaultDialog THEN
	GVL_MASTER.stAlarms[0].aEventFlags[46] := TRUE;
END_IF


//Remove Nest **LA 17092025
IF GVL_HMI_GLOBAL.bStartButton AND NOT PRG_Mastercycle.biClamp AND PRG_Mastercycle.biPartPresent THEN 
	GVL_MASTER.stAlarms[0].aEventFlags[100] := TRUE;
	ELSIF NOT PRG_Mastercycle.biPartPresent THEN 
		GVL_MASTER.stAlarms[0].aEventFlags[100] := FALSE;
END_IF

//Release Clamp  **LA 17092025
IF GVL_HMI_GLOBAL.bStartButton AND PRG_Mastercycle.biClamp AND NOT PRG_Mastercycle.biPartPresent AND GVL_MASTER.stMachineStatus.bSystemReadyToStart THEN 
	GVL_MASTER.stAlarms[0].aEventFlags[101] := TRUE;
	ELSIF NOT PRG_Mastercycle.biClamp THEN 
		GVL_MASTER.stAlarms[0].aEventFlags[101] := FALSE;
END_IF

//Releas Clamp and Remove Nest  **LA 17092025
IF GVL_HMI_GLOBAL.bStartButton AND PRG_Mastercycle.biClamp AND PRG_Mastercycle.biPartPresent AND GVL_MASTER.stMachineStatus.bSystemReadyToStart THEN
	GVL_MASTER.stAlarms[0].aEventFlags[102] := TRUE;
	ELSIF  NOT PRG_Mastercycle.biClamp AND NOT PRG_Mastercycle.biPartPresent THEN
		GVL_MASTER.stAlarms[0].aEventFlags[102] := FALSE;
END_IF
END_ACTION

METHOD PRIVATE SetEventTexts : BOOL
VAR_INPUT
END_VAR
//Immediate Faults
GVL_MASTER.stAlarms[0].aEventTexts[0] := 'SPARE';
GVL_MASTER.stAlarms[0].aEventTexts[1] := 'SPARE';
GVL_MASTER.stAlarms[0].aEventTexts[2] := 'SPARE';
GVL_MASTER.stAlarms[0].aEventTexts[3] := 'SPARE';
GVL_MASTER.stAlarms[0].aEventTexts[4] := '';
GVL_MASTER.stAlarms[0].aEventTexts[5] := '';
GVL_MASTER.stAlarms[0].aEventTexts[6] := '';
GVL_MASTER.stAlarms[0].aEventTexts[7] := '';
GVL_MASTER.stAlarms[0].aEventTexts[8] := '';
GVL_MASTER.stAlarms[0].aEventTexts[9] := '';
GVL_MASTER.stAlarms[0].aEventTexts[10] := '';
GVL_MASTER.stAlarms[0].aEventTexts[10] := ''; 
GVL_MASTER.stAlarms[0].aEventTexts[11] := '';
GVL_MASTER.stAlarms[0].aEventTexts[12] := '';
GVL_MASTER.stAlarms[0].aEventTexts[13] := '';
GVL_MASTER.stAlarms[0].aEventTexts[14] := '';
GVL_MASTER.stAlarms[0].aEventTexts[15] := '';


//Cycle stop fault

GVL_MASTER.stAlarms[0].aEventTexts[33] := 'Beckhoff EL1809 Not Operational';
GVL_MASTER.stAlarms[0].aEventTexts[34] := 'Beckhoff EL2809 Not Operational';
GVL_MASTER.stAlarms[0].aEventTexts[35] := 'Cognex  IS2801M Connection Error';
GVL_MASTER.stAlarms[0].aEventTexts[36] := 'External Error - Cognex Camera ERROR';
GVL_MASTER.stAlarms[0].aEventTexts[37] := 'Cognex  IS2801M Diagnostic Error';
GVL_MASTER.stAlarms[0].aEventTexts[38] := 'Master - Stopping timeout';
GVL_MASTER.stAlarms[0].aEventTexts[39] := 'User Not Log IN';
GVL_MASTER.stAlarms[0].aEventTexts[40] := 'User Log-Off Timeout Manual Mode'; 
GVL_MASTER.stAlarms[0].aEventTexts[41] := 'Keyence DL-P1 Error';
GVL_MASTER.stAlarms[0].aEventTexts[42] := 'Autocyle Timeou' ;
GVL_MASTER.stAlarms[0].aEventTexts[43] := 'Part removed during cycle';
GVL_MASTER.stAlarms[0].aEventTexts[44] := 'Clamp toggled before requested';
GVL_MASTER.stAlarms[0].aEventTexts[45] := 'Clamp toggled before requested';
GVL_MASTER.stAlarms[0].aEventTexts[46] := 'Press Acknowledge';
GVL_MASTER.stAlarms[0].aEventTexts[47] := '';
GVL_MASTER.stAlarms[0].aEventTexts[48] := '';
GVL_MASTER.stAlarms[0].aEventTexts[59] := '';
GVL_MASTER.stAlarms[0].aEventTexts[50] := '';

//Cycle Stop Requests

GVL_MASTER.stAlarms[0].aEventTexts[80] := 'Machine Cycle Stop 10 Min Not Use Timeout';
GVL_MASTER.stAlarms[0].aEventTexts[81] := '';
GVL_MASTER.stAlarms[0].aEventTexts[82] := '';

GVL_MASTER.stAlarms[0].aEventTexts[84] := '';
GVL_MASTER.stAlarms[0].aEventTexts[85] := '';
GVL_MASTER.stAlarms[0].aEventTexts[86] := '';
GVL_MASTER.stAlarms[0].aEventTexts[87] := ''; 
GVL_MASTER.stAlarms[0].aEventTexts[88] := '';
GVL_MASTER.stAlarms[0].aEventTexts[89] := '';


// Message //**LA 15092025
GVL_MASTER.stAlarms[0].aEventTexts[100] := 'Remove Nest';
GVL_MASTER.stAlarms[0].aEventTexts[101] := 'Release Clamp';
GVL_MASTER.stAlarms[0].aEventTexts[102] := 'Release Clamp and Remove Nest';
END_METHOD

END_PROGRAM

// ---- POUs/A_Master/PRG_MasterCycle.TcPOU
PROGRAM PRG_MasterCycle
VAR
	
		tonCaseTimDelay    	: ARRAY [1..20] OF Tc2_Standard.TON;
	    rtrigCaseTriger    	: ARRAY [1..10] OF Tc2_Standard.R_TRIG;
		ftrigCaseTriger		: ARRAY [1..10] OF Tc2_Standard.F_TRIG;
	   	rtrigFaultMachine  	: Tc2_Standard.R_TRIG;	
		
		biClamp				: BOOL;
		biPartPresent		: BOOL;
		


		bAutoCycleStop		: BOOL;
		
		bCycleFlag			: BOOL;
		bGreenLED			: BOOL;
		bRedLED				: BOOL;
		bEndCycleFlag		: BOOL;
		bStationsStopped	: BOOL;
		bHeighTestCompleteFlag : BOOL;
		bLeakTestCompleteFlag : BOOL;
		i					: DINT;
		
		


END_VAR
VAR_IN_OUT
	stStationStruct          : ST_StandardStationStruct;
END_VAR

ACT_LinkIO();
ACT_TimTrig();
stStationStruct.bStationInProgress := stStationStruct.nState>=1100 AND stStationStruct.nState<=1600;

IF stStationStruct.nState <700 OR  stStationStruct.nState > 4000 THEN
	GVL_HMI_GLOBAL.sActualProcess := ""; 
	GVL_MASTER.stNest.bPiecePass 	:= FALSE;
	GVL_MASTER.stNest.bPieceReject 	:= FALSE;
	bGreenLED						:= FALSE;
	bRedLED							:= FALSE;
	GVL_MASTER.stNest.bHeightPass 	:= FALSE;
	GVL_MASTER.stNest.bLeakPass 	:= FALSE;
	GVL_MASTER.stNest.bVisionPass 	:= FALSE;
	GVL_MASTER.stNest.bHeightReject := FALSE;
	GVL_MASTER.stNest.bLeakReject	:= FALSE;
	GVL_MASTER.stNest.bVisionReject := FALSE;
END_IF

IF rtrigCaseTriger[3].Q THEN
GVL_PERSIST.stPartsInspection.nPartsGood:= GVL_PERSIST.stPartsInspection.nPartsGood +1;
GVL_PERSIST.stPartsInspection.nTotalPartsGood := GVL_PERSIST.stPartsInspection.nTotalPartsGood+1;
ELSIF GVL_HMI_GLOBAL.bResetGoodParts THEN
GVL_PERSIST.stPartsInspection.nPartsGood:=0;	
END_IF


IF rtrigCaseTriger[4].Q THEN
	GVL_PERSIST.stPartsInspection.nPartsFailed:=GVL_PERSIST.stPartsInspection.nPartsFailed+1;
	GVL_PERSIST.stPartsInspection.nTotalPartsFailed:= GVL_PERSIST.stPartsInspection.nTotalPartsFailed+1;
ELSIF GVL_HMI_GLOBAL.bResetFailedParts THEN
	GVL_PERSIST.stPartsInspection.nPartsFailed:=0;
END_IF

IF stStationStruct.nState < 700 THEN
	 GVL_HMI_GLOBAL.sMessageToOperator := "Press Reset Button to Home Machine";
END_IF

CASE stStationStruct.nState OF
	
100: 
   bAutoCycleStop := FALSE;
IF NOT GVL_MASTER.stMachineStatus.bSystemPowerUp THEN
	stStationStruct.nState := 200;
END_IF
200:
IF GVL_MASTER.stMachineStatus.bSystemInitialising THEN
	stStationStruct.nState := 300;
END_IF
300:
   GVL_Master.stStationSruct[1].bStationInitRequest := TRUE;
   GVL_Master.stStationSruct[2].bStationInitRequest := TRUE;
   GVL_Master.stStationSruct[3].bStationInitRequest := TRUE;
   
IF GVL_Master.stStationSruct[1].bStationInitRequest AND GVL_Master.stStationSruct[2].bStationInitRequest AND
   GVL_Master.stStationSruct[3].bStationInitRequest  THEN
	stStationStruct.nState := 400;
END_IF
400:
IF NOT GVL_Master.stStationSruct[1].bStationInitRequest AND NOT GVL_Master.stStationSruct[2].bStationInitRequest AND
   NOT GVL_Master.stStationSruct[3].bStationInitRequest THEN
	stStationStruct.nState := 500;   
END_IF 
500:
   GVL_Master.stStationSruct[1].bStationAcknowledge := TRUE;
   GVL_Master.stStationSruct[2].bStationAcknowledge := TRUE;
   GVL_Master.stStationSruct[3].bStationAcknowledge := TRUE;
IF   GVL_Master.stStationSruct[1].bStationAcknowledge AND  GVL_Master.stStationSruct[2].bStationAcknowledge AND
     GVL_Master.stStationSruct[3].bStationAcknowledge THEN
     stStationStruct.nState := 600;
END_IF
600:
IF GVL_Master.stStationSruct[1].bStationHomed AND GVL_Master.stStationSruct[2].bStationHomed AND GVL_Master.stStationSruct[3].bStationHomed  THEN
   GVL_Master.stStationSruct[1].bStationAcknowledge := FALSE;
   GVL_Master.stStationSruct[2].bStationAcknowledge := FALSE;
   GVL_Master.stStationSruct[3].bStationAcknowledge := FALSE;
   stStationStruct.nState := 700;
END_IF
700: // All Station Homed and waiting for Autocycle 
   bAutoCycleStop := FALSE;
   GVL_HMI_GLOBAL.sActualProcess := "Waiting for Autocycle";
   IF GVL_MASTER.stMachineStatus.bSystemReadyToStart THEN 
	  GVL_HMI_GLOBAL.sMessageToOperator := "Press Start Button to Autocycle";
   ELSE GVL_HMI_GLOBAL.sMessageToOperator := "Press Reset Button to Reset machine";
   END_IF
   
IF GVL_Master.stMachineStatus.bSystemAutoCycle THEN
	stStationStruct.nState := 800;
ELSIF GVL_Master.stMachineStatus.bManualMode THEN
      stStationStruct.nState := 4000;
ELSIF GVL_Master.stMachineStatus.bSystemStopping AND NOT bStationsStopped  THEN
      stStationStruct.nState := 5000;
ELSIF GVL_Master.stMachineStatus.bCycleStopFault OR GVL_Master.stMachineStatus.bImmediateFault THEN
      stStationStruct.nState := 6000;	  
END_IF

IF tonCaseTimDelay[9].Q THEN
	stStationStruct.nState := 1000;
END_IF
800:
stStationStruct.nState := 1000;
1000: // System Autocycle

IF biPartPresent THEN
	GVL_HMI_GLOBAL.sMessageToOperator := "Remove Nest";
ELSE GVL_HMI_GLOBAL.sMessageToOperator := "Insert Nest to begin process";
END_IF


IF  rtrigCaseTriger [5].Q  AND NOT bEndCycleFlag THEN
	GVL_MASTER.stNest.bHeightPass 	:= FALSE;
	GVL_MASTER.stNest.bLeakPass 	:= FALSE;
	GVL_MASTER.stNest.bVisionPass 	:= FALSE;
	GVL_MASTER.stNest.bHeightReject := FALSE;
	GVL_MASTER.stNest.bLeakReject	:= FALSE;
	GVL_MASTER.stNest.bVisionReject := FALSE;
	GVL_MASTER.stNest.bPiecePass 	:= FALSE;
	GVL_MASTER.stNest.bPieceReject 	:= FALSE;
	GVL_MASTER.stNest.bNestPartProced := FALSE;
	GVL_MASTER.stNest.sHeightHMI 	:= "";
	GVL_MASTER.stNest.sLeakHMI 		:= "";
	GVL_MASTER.stNest.sVisionHMI 	:= "";
	GVL_MASTER.stNest.sPieceHMI 	:= "";
	bCycleFlag						:= TRUE;
	GVL_HMI_GLOBAL.sMessageToOperator := "Process in progress";
	GVL_HMI_GLOBAL.bResetPassAndFail:= TRUE;
	GVL_HMI_GLOBAL.sActualProcess := "";
	bGreenLED						:= FALSE;
	bRedLED							:= FALSE;
	GVL_HMI_GLOBAL.bRejectPieceAcknowledge := FALSE;
	stStationStruct.nState 			:= 1130;
	
ELSIF GVL_Master.stMachineStatus.bSystemStopping  THEN
      stStationStruct.nState := 5000;
ELSIF tonCaseTimDelay[10].Q THEN
	  bAutoCycleStop := TRUE;
      stStationStruct.nState := 5000;	
END_IF
1130:
IF tonCaseTimDelay[13].Q THEN
	GVL_HMI_GLOBAL.bResetPassAndFail:= FALSE;
	stStationStruct.nState 			:= 1132;
END_IF


//Vision Test
1132: 
	GVL_MASTER.anValueBeforeMeasurement := GVL_MASTER.aSensorCurrentValue;
	GVL_HMI_GLOBAL.sActualProcess := "Vision process"; 
	GVL_Master.stStationSruct[3].bStationRequest := TRUE;
	stStationStruct.nState := 1134;
1134:
IF GVL_Master.stStationSruct[3].bStationInProgress THEN
	stStationStruct.nState := 1136;
END_IF
1136:
IF GVL_Master.stStationSruct[3].bStationComplete AND NOT GVL_Master.stMachineStatus.bSystemStopping THEN
	stStationStruct.nState := 1138;
ELSIF GVL_Master.stMachineStatus.bSystemStopping OR ftrigCaseTriger [1].Q THEN
	stStationStruct.nState := 5000;
END_IF
1138:
GVL_HMI_GLOBAL.sMessageToOperator := "Toggle Clamp to continue the process";
IF rtrigCaseTriger [1].Q  THEN
	stStationStruct.nState := 1142;
ELSIF GVL_Master.stMachineStatus.bSystemStopping  THEN
      stStationStruct.nState := 5000;
ELSIF tonCaseTimDelay[10].Q THEN
	  bAutoCycleStop := TRUE;
      stStationStruct.nState := 5000;	

END_IF
//Leak test
1142: 
	GVL_HMI_GLOBAL.sMessageToOperator := "Process in progress";
	GVL_HMI_GLOBAL.sActualProcess := "Leak And Height test process"; 
	GVL_Master.stStationSruct[2].bStationRequest := TRUE;
	GVL_Master.stStationSruct[1].bStationRequest := TRUE;
	stStationStruct.nState := 1144;
1144:
IF GVL_Master.stStationSruct[2].bStationInProgress AND GVL_Master.stStationSruct[1].bStationInProgress THEN
	stStationStruct.nState := 1146;
END_IF
1146:
IF GVL_Master.stStationSruct[2].bStationComplete THEN
	bHeighTestCompleteFlag := TRUE;
END_IF
IF GVL_Master.stStationSruct[1].bStationComplete THEN
	bLeakTestCompleteFlag := TRUE;
END_IF

IF bHeighTestCompleteFlag AND bLeakTestCompleteFlag AND NOT GVL_Master.stMachineStatus.bSystemStopping THEN
	stStationStruct.nState := 1152;
	GVL_MASTER.bHeightTestacknowledge := TRUE;
ELSIF GVL_Master.stMachineStatus.bSystemStopping THEN
	stStationStruct.nState := 5000;
END_IF

1152: 
	GVL_MASTER.stNest.bNestPartProced 	:= TRUE;
	bHeighTestCompleteFlag				:= FALSE;
	bLeakTestCompleteFlag				:= FALSE;
IF tonCaseTimDelay[12].Q THEN
	GVL_MASTER.bHeightTestacknowledge := FALSE;
	stStationStruct.nState := 1220;
END_IF
	
1220:
IF GVL_MASTER.stNest.bHeightPass AND GVL_MASTER.stNest.bLeakPass AND GVL_MASTER.stNest.bVisionPass THEN
	GVL_MASTER.stNest.bPiecePass 	:= TRUE;
	GVL_MASTER.stNest.bPieceReject 	:= FALSE;
	GVL_MASTER.stNest.sPieceHMI 	:= "Pass";
	bGreenLED						:= TRUE;
	bRedLED							:= FALSE;
ELSE GVL_MASTER.stNest.bNestPartOK := FALSE;
	GVL_MASTER.stNest.sPieceHMI 	:= "Fail";
	GVL_MASTER.stNest.bPiecePass 	:= FALSE;
	GVL_MASTER.stNest.bPieceReject 	:= TRUE;
	bGreenLED						:= FALSE;
	bRedLED							:= TRUE;
END_IF
GVL_MASTER.stNest.sDate := GVL_HMI_GLOBAL.sSystemDate;
GVL_MASTER.stNest.sTime := GVL_HMI_GLOBAL.sSystemTime;

IF rtrigCaseTriger [8].Q THEN	
	
	FOR i :=200 TO 2 BY (-1) DO
		GVL_HMI_GLOBAL.aStatistics[i]	:= GVL_HMI_GLOBAL.aStatistics[i-1];
	END_FOR
	
	GVL_HMI_GLOBAL.aStatistics[1] := GVL_MASTER.stNest;
END_IF

IF tonCaseTimDelay[11].Q THEN
	stStationStruct.nState := 1500;
END_IF

1500:
IF GVL_Master.stStationSruct[1].bStationNotMoving AND GVL_Master.stStationSruct[2].bStationNotMoving AND GVL_Master.stStationSruct[3].bStationNotMoving THEN
	stStationStruct.nState := 1550;
END_IF
1550:
IF  GVL_MASTER.stNest.bPiecePass THEN	
	stStationStruct.nState := 1600;
ELSIF  GVL_MASTER.stNest.bPieceReject AND GVL_HMI_GLOBAL.bRejectPieceAcknowledge THEN
	stStationStruct.nState := 1600;
END_IF

1600:
GVL_HMI_GLOBAL.sMessageToOperator 				:= "Cycle Complete";   // **LAA 17092025
bEndCycleFlag	:= TRUE;
IF NOT GVL_MASTER.stMachineStatus.bSystemStopping  THEN 
	stStationStruct.nState := 1700;
ELSE 
    stStationStruct.nState := 5000;	
END_IF
1700:
GVL_HMI_GLOBAL.sMessageToOperator 				:= "Release Clamp";    // **LAA 17092025
IF rtrigCaseTriger [7].Q  THEN 
	stStationStruct.nState := 1000; 
END_IF

4000: 
IF NOT GVL_MASTER.stMachineStatus.bManualMode THEN
	stStationStruct.nState := 700;	
ELSIF GVL_MASTER.stMachineStatus.bCycleStopFault OR GVL_MASTER.stMachineStatus.bImmediateFault THEN
      stStationStruct.nState := 6000;		
END_IF

//stopping
5000:
	GVL_Master.stStationSruct[1].bNoCycleStopRequest := FALSE;
    GVL_Master.stStationSruct[2].bNoCycleStopRequest := FALSE;
	GVL_Master.stStationSruct[3].bNoCycleStopRequest := FALSE;
	

IF tonCaseTimDelay[6].Q AND (GVL_Master.stStationSruct[1].nState = 1000) AND (GVL_Master.stStationSruct[2].nState = 1000) 
                        AND (GVL_Master.stStationSruct[3].nState = 1000) THEN
	bAutoCycleStop := FALSE;
	
	stStationStruct.nState := 700;

	
END_IF

6000:
IF tonCaseTimDelay[1].Q THEN
	GVL_Master.stStationSruct[1].bStationInitRequest := FALSE;
	GVL_Master.stStationSruct[2].bStationInitRequest := FALSE;
	GVL_Master.stStationSruct[3].bStationInitRequest := FALSE;
	GVL_Master.stStationSruct[1].bStationRequest := FALSE;
	GVL_Master.stStationSruct[2].bStationRequest := FALSE;
    GVL_Master.stStationSruct[3].bStationRequest := FALSE;
	GVL_Master.stStationSruct[1].bStationAbort := TRUE;
    GVL_Master.stStationSruct[2].bStationAbort := TRUE;
	GVL_Master.stStationSruct[3].bStationAbort := TRUE;
	stStationStruct.nState := 100;
END_IF


END_CASE

//++++++++++++++++++++++++++++++++++++++++++++++++++++++++++++++++++++++++++++++++++++++++++++++++++++++++++++++++++++++++++++++++++++++

IF rtrigFaultMachine.Q THEN
   stStationStruct.nState := 6000;	  
END_IF

IF  (stStationStruct.nState = 4000) OR (stStationStruct.nState = 5000) OR (stStationStruct.nState = 6000) THEN
   GVL_Master.stStationSruct[1].bStationAcknowledge := FALSE;
   GVL_Master.stStationSruct[2].bStationAcknowledge := FALSE;
   GVL_Master.stStationSruct[3].bStationAcknowledge := FALSE;
   GVL_Master.stStationSruct[1].bStationInitRequest := FALSE;
   GVL_Master.stStationSruct[2].bStationInitRequest := FALSE;
   GVL_Master.stStationSruct[3].bStationInitRequest := FALSE;
END_IF

ACTION ACT_LinkIO:
// Initialisation Progres
IF GVL_Master.stStationSruct[1].bStationInProgressInit THEN
	GVL_Master.stStationSruct[1].bStationInitRequest := FALSE;
END_IF
IF GVL_Master.stStationSruct[2].bStationInProgressInit THEN
	GVL_Master.stStationSruct[2].bStationInitRequest := FALSE;
END_IF
IF GVL_Master.stStationSruct[3].bStationInProgressInit THEN
	GVL_Master.stStationSruct[3].bStationInitRequest := FALSE;
END_IF

// Cycle Progres
IF GVL_Master.stStationSruct[1].bStationInProgress THEN
	GVL_Master.stStationSruct[1].bStationRequest := FALSE;
END_IF
IF GVL_Master.stStationSruct[2].bStationInProgress THEN
	GVL_Master.stStationSruct[2].bStationRequest := FALSE;
END_IF
IF GVL_Master.stStationSruct[3].bStationInProgress THEN
	GVL_Master.stStationSruct[3].bStationRequest := FALSE;
END_IF

// Abort Station
IF GVL_Master.stStationSruct[1].nState = 100 THEN
	GVL_Master.stStationSruct[1].bStationAbort := FALSE;
END_IF
IF GVL_Master.stStationSruct[2].nState = 100 THEN	
    GVL_Master.stStationSruct[2].bStationAbort := FALSE;
END_IF	
IF GVL_Master.stStationSruct[3].nState = 100 THEN
	GVL_Master.stStationSruct[3].bStationAbort := FALSE;
END_IF

IF (GVL_Master.stStationSruct[1].nState = 100) OR (GVL_Master.stStationSruct[1].nState = 1000) THEN
	GVL_Master.stStationSruct[1].bNoCycleStopRequest := TRUE;
END_IF
IF (GVL_Master.stStationSruct[2].nState = 100) OR (GVL_Master.stStationSruct[2].nState = 1000) THEN	
    GVL_Master.stStationSruct[2].bNoCycleStopRequest := TRUE;
END_IF
IF (GVL_Master.stStationSruct[3].nState = 100) OR (GVL_Master.stStationSruct[3].nState = 1000) THEN	
	GVL_Master.stStationSruct[3].bNoCycleStopRequest := TRUE;
END_IF

IF  (GVL_Master.stStationSruct[1].nState = 1000) AND (GVL_Master.stStationSruct[2].nState = 1000) 
                        AND (GVL_Master.stStationSruct[3].nState = 1000) THEN
	bStationsStopped := TRUE;
ELSE bStationsStopped := FALSE;

END_IF

GVL_MASTER.stMasterControl.bAllStationsCycledStopped := (GVL_Master.stStationSruct[1].nState = 1000) AND (GVL_Master.stStationSruct[2].nState = 1000) 
                                         AND (GVL_Master.stStationSruct[3].nState = 1000)
										 AND  stStationStruct.nState=700;
										 
	biClamp									:= GVL_IO.dw_T02_EL1809.iCalmpClosed;
	biPartPresent							:=  GVL_IO.dw_T02_EL1809.iPartPresent;
	GVL_MASTER.stNest.bNestPresent			:= GVL_IO.dw_T02_EL1809.iCalmpClosed;
	GVL_IO.dw_T03_EL2809.qPassIndicatorGreen:= bGreenLED;
	GVL_IO.dw_T03_EL2809.qRejectIndicatorRed:= bRedLED;
	
IF ftrigCaseTriger[1].Q THEN
	bEndCycleFlag							:= FALSE;
END_IF
	
GVL_MASTER.aSensorCurrentValue[1] 					:= GVL_IO.dw_B08_DL_PN1.gt2_1_1CurrentValue;
GVL_MASTER.aSensorCurrentValue[2] 					:= GVL_IO.dw_B08_DL_PN1.gt2_1_2CurrentValue;
GVL_MASTER.aSensorCurrentValue[3] 					:= GVL_IO.dw_B08_DL_PN1.gt2_1_3CurrentValue;
GVL_MASTER.aSensorCurrentValue[4] 					:= GVL_IO.dw_B08_DL_PN1.gt2_2CurrentValue;
END_ACTION

ACTION ACT_TimTrig:
tonCaseTimDelay[1](IN:= (stStationStruct.nState = 6000),PT:=T#100MS); //
tonCaseTimDelay[2](IN:= (stStationStruct.nState = 5000),PT:=T#100MS); //
tonCaseTimDelay[3](IN:= (stStationStruct.nState = 1100),PT:=T#40MS);  //
tonCaseTimDelay[4](IN:= (stStationStruct.nState = 1140),PT:=T#250MS);
tonCaseTimDelay[5](IN:= (stStationStruct.nState = 1900),PT:=T#250MS);
tonCaseTimDelay[6](IN:= (stStationStruct.nState = 5000),PT:=T#250MS);
tonCaseTimDelay[7](IN:= (stStationStruct.nState = 1340),PT:=T#200MS);
tonCaseTimDelay[8](IN:= (stStationStruct.nState = 1320),PT:=T#500MS);
tonCaseTimDelay[9](IN:= (stStationStruct.nState = 800),PT:=T#3S);
tonCaseTimDelay[10](IN:= (stStationStruct.nState = 1000),PT:=T#10M);
tonCaseTimDelay[11](IN:= (stStationStruct.nState = 1220),PT:=T#1S);
tonCaseTimDelay[12](IN:= stStationStruct.nState = 1152,PT:=T#1S );
tonCaseTimDelay[13](IN:=(stStationStruct.nState = 1130),PT:=T#1S );
tonCaseTimDelay[14](IN:=,PT:=T#1S);
tonCaseTimDelay[15](IN:= );
tonCaseTimDelay[16](IN:= );
tonCaseTimDelay[17](IN:= );
tonCaseTimDelay[18](IN:= );
tonCaseTimDelay[19](IN:= );
tonCaseTimDelay[20](IN:= );

rtrigCaseTriger [1](CLK:= biClamp);
rtrigCaseTriger [2](CLK:= tonCaseTimDelay[2].Q);
rtrigCaseTriger [3](CLK:= GVL_MASTER.stNest.bPiecePass);
rtrigCaseTriger [4](CLK:= GVL_MASTER.stNest.bPieceReject);
rtrigCaseTriger [5](CLK:= biPartPresent );
rtrigCaseTriger [6](CLK:= );
rtrigCaseTriger [7](CLK:= NOT biClamp);  // **LAA 17092025);
rtrigCaseTriger [8](CLK:= stStationStruct.nState = 1220);
rtrigCaseTriger [9](CLK:= );
rtrigCaseTriger [10](CLK:= );
rtrigFaultMachine(CLK:= GVL_MASTER.stMachineStatus.bCycleStopFault OR GVL_MASTER.stMachineStatus.bImmediateFault);

ftrigCaseTriger [1](CLK:= biPartPresent );
END_ACTION

END_PROGRAM

// ---- POUs/B_HightTest/PRG_Fault_HeightTest.TcPOU
PROGRAM PRG_Fault_HeightTest
VAR
	
			i					: INT;
END_VAR
VAR_IN_OUT

  aAlarms  : ARRAY[0..3] OF ST_Events;
END_VAR

ACT_FaultTrig();

(************************************** Faults reset **********************************************)
IF   GVL_HMI_GLOBAL.bResetButton THEN 
	FOR i := 0 TO 127 DO
		GVL_MASTER.stAlarms[1].aEventFlags[i] := FALSE;
	END_FOR
END_IF
//===============================================================
//Initialize event texts on first scan
IF NOT GVL_MASTER.stAlarms[1].bEventTextsSet THEN
	SetEventTexts();
	GVL_MASTER.stAlarms[1].bEventTextsSet := TRUE;
END_IF


(***************************************************************************************************)
//Immediate fault
GVL_MASTER.stAlarms[1].bImmediateFault := FALSE;
FOR i := 0 TO 32DO
	GVL_MASTER.stAlarms[1].bImmediateFault := GVL_MASTER.stAlarms[1].bImmediateFault OR GVL_MASTER.stAlarms[1].aEventFlags[i];
END_FOR

//Cycle stop fault
GVL_MASTER.stAlarms[1].bCycleStopFault := FALSE;
FOR i := 33 TO 79 DO
	GVL_MASTER.stAlarms[1].bCycleStopFault := GVL_MASTER.stAlarms[1].bCycleStopFault OR GVL_MASTER.stAlarms[1].aEventFlags[i];
END_FOR

//Cycle stop REQUEST
GVL_MASTER.stAlarms[1].bCycleStopRequest := FALSE;
FOR i := 80 TO 99 DO
	GVL_MASTER.stAlarms[1].bCycleStopRequest := GVL_MASTER.stAlarms[1].bCycleStopRequest OR GVL_MASTER.stAlarms[1].aEventFlags[i];
END_FOR

ACTION ACT_FaultTrig:
(**************************************************************************************************)
(**************************** Master Immediate Fault Stop *****************************************)
(**************************************************************************************************)
(* Copy Safety Immediate Stop Faults to Master Immediate Stop Faults *)
(* *)

//Station 3 - Keyence Inspection Homing Time Out
GVL_MASTER.stAlarms[1].aEventTimers[1](IN := (GVL_MASTER.stStationSruct[1].nState>=200 AND GVL_MASTER.stStationSruct[1].nState<=900),PT:= T#10000MS );
IF GVL_MASTER.stAlarms[1].aEventTimers[1].Q  THEN // Fault 1
	GVL_MASTER.stAlarms[1].aEventFlags[1] := TRUE;
END_IF
// Probe 1 Current Value Invalid
GVL_MASTER.stAlarms[1].aEventTimers[2](IN:= GVL_IO.dw_B08_DL_PN1.gt2_1_1CurrValInv ,PT:= T#100MS);
IF GVL_MASTER.stAlarms[1].aEventTimers[2].Q  THEN // Fault 2
	GVL_MASTER.stAlarms[1].aEventFlags[2] := TRUE;
END_IF
// Probe 2 Current Value Invalid
GVL_MASTER.stAlarms[1].aEventTimers[3](IN:= GVL_IO.dw_B08_DL_PN1.gt2_1_2CurrValInv ,PT:= T#100MS);
IF GVL_MASTER.stAlarms[1].aEventTimers[3].Q  THEN // Fault 3
	GVL_MASTER.stAlarms[1].aEventFlags[3] := TRUE;
END_IF
// Probe 3 Current Value Invalid
GVL_MASTER.stAlarms[1].aEventTimers[4](IN:= GVL_IO.dw_B08_DL_PN1.gt2_1_3CurrValInv ,PT:= T#100MS);
IF GVL_MASTER.stAlarms[1].aEventTimers[4].Q  THEN // Fault 4
	GVL_MASTER.stAlarms[1].aEventFlags[4] := TRUE;
END_IF
// Probe 4 Current Value Invalid
GVL_MASTER.stAlarms[1].aEventTimers[5](IN:= GVL_IO.dw_B08_DL_PN1.gt2_2CurrValInv ,PT:= T#100MS);
IF GVL_MASTER.stAlarms[1].aEventTimers[5].Q  THEN // Fault 5
	GVL_MASTER.stAlarms[1].aEventFlags[5] := TRUE;
END_IF
// Probe 1 Error
GVL_MASTER.stAlarms[1].aEventTimers[6](IN:= GVL_IO.dw_B08_DL_PN1.gt2_1_1ErrorStat ,PT:= T#100MS);
IF GVL_MASTER.stAlarms[1].aEventTimers[6].Q  THEN // Fault 6
	GVL_MASTER.stAlarms[1].aEventFlags[6] := TRUE;
END_IF
// Probe 2 Error
GVL_MASTER.stAlarms[1].aEventTimers[7](IN:= GVL_IO.dw_B08_DL_PN1.gt2_1_2ErrorStat  ,PT:= T#100MS);
IF GVL_MASTER.stAlarms[1].aEventTimers[7].Q  THEN // Fault 7
	GVL_MASTER.stAlarms[1].aEventFlags[7] := TRUE;
END_IF
// Probe 3 Error
GVL_MASTER.stAlarms[1].aEventTimers[8](IN:= GVL_IO.dw_B08_DL_PN1.gt2_1_3ErrorStat  ,PT:= T#100MS);
IF GVL_MASTER.stAlarms[1].aEventTimers[8].Q  THEN // Fault 8
	GVL_MASTER.stAlarms[1].aEventFlags[8] := TRUE;
END_IF
// Probe 4 Error
GVL_MASTER.stAlarms[1].aEventTimers[9](IN:= GVL_IO.dw_B08_DL_PN1.gt2_1_1ErrorStat  ,PT:= T#100MS);
IF GVL_MASTER.stAlarms[1].aEventTimers[9].Q  THEN // Fault 9
	GVL_MASTER.stAlarms[1].aEventFlags[9] := TRUE;
END_IF

// Master Probe Error
GVL_MASTER.stAlarms[1].aEventTimers[10](IN:= GVL_IO.dw_B08_DL_PN1.dldErrorStt ,PT:= T#100MS);
IF GVL_MASTER.stAlarms[1].aEventTimers[10].Q  THEN // Fault 10
	GVL_MASTER.stAlarms[1].aEventFlags[10] := TRUE;
END_IF

//Height Station Cycle Timeout
GVL_MASTER.stAlarms[1].aEventTimers[11](IN:= (GVL_Master.stStationSruct[1].nState>=1100 AND GVL_Master.stStationSruct[1].nState<=1900) ,PT:=T#10S);
IF GVL_MASTER.stAlarms[1].aEventTimers[11].Q THEN // 
	GVL_MASTER.stAlarms[1].aEventFlags[11] := TRUE;
END_IF
// Sensor 1 Stuck
IF GVL_MASTER.abSensorStuck[1]  THEN 
	GVL_MASTER.stAlarms[1].aEventFlags[12] := TRUE;
END_IF
// Sensor 2 Stuck
IF GVL_MASTER.abSensorStuck[2]  THEN 
	GVL_MASTER.stAlarms[1].aEventFlags[13] := TRUE;
END_IF
// Sensor 3 Stuck
IF GVL_MASTER.abSensorStuck[3]  THEN 
	GVL_MASTER.stAlarms[1].aEventFlags[14] := TRUE;
END_IF
// Sensor 4 Stuck
IF GVL_MASTER.abSensorStuck[4]  THEN 
	GVL_MASTER.stAlarms[1].aEventFlags[15] := TRUE;
END_IF
END_ACTION

METHOD PRIVATE SetEventTexts : BOOL
VAR_INPUT
END_VAR
//Immediate Faults
GVL_MASTER.stAlarms[1].aEventTexts[0] := '';
GVL_MASTER.stAlarms[1].aEventTexts[1] := 'Station 3 - Keyence Inspection Homing Time Out';
GVL_MASTER.stAlarms[1].aEventTexts[2] := 'Invalid Value Probe 1';
GVL_MASTER.stAlarms[1].aEventTexts[3] := 'Invalid Value Probe 2';
GVL_MASTER.stAlarms[1].aEventTexts[4] := 'Invalid Value Probe 3';
GVL_MASTER.stAlarms[1].aEventTexts[5] := 'Invalid Value Probe 4';
GVL_MASTER.stAlarms[1].aEventTexts[6] := 'Error State Probe 1';
GVL_MASTER.stAlarms[1].aEventTexts[7] := 'Error State Probe 2';
GVL_MASTER.stAlarms[1].aEventTexts[8] := 'Error State Probe 3';
GVL_MASTER.stAlarms[1].aEventTexts[9] := 'Error State Probe 4'; 
GVL_MASTER.stAlarms[1].aEventTexts[10] := 'Error Master Probes Profinet'; 
GVL_MASTER.stAlarms[1].aEventTexts[11] := 'Height Station Cycle Timeout';
GVL_MASTER.stAlarms[1].aEventTexts[12] := 'Sensor 1 Stuck';
GVL_MASTER.stAlarms[1].aEventTexts[13] := 'Sensor 2 Stuck';
GVL_MASTER.stAlarms[1].aEventTexts[14] := 'Sensor 3 Stuck';
GVL_MASTER.stAlarms[1].aEventTexts[15] := 'Sensor 4 Stuck';
GVL_MASTER.stAlarms[1].aEventTexts[16] := '';
GVL_MASTER.stAlarms[1].aEventTexts[17] := '';
GVL_MASTER.stAlarms[1].aEventTexts[18] := '';
GVL_MASTER.stAlarms[1].aEventTexts[19] := '';
GVL_MASTER.stAlarms[1].aEventTexts[20] := '';
GVL_MASTER.stAlarms[1].aEventTexts[21] := '';
GVL_MASTER.stAlarms[1].aEventTexts[22] := '';
GVL_MASTER.stAlarms[1].aEventTexts[28] := '';
GVL_MASTER.stAlarms[1].aEventTexts[29] := '';
GVL_MASTER.stAlarms[1].aEventTexts[30] := '';

//Cycle Stop Requests

GVL_MASTER.stAlarms[1].aEventTexts[80] := '';
GVL_MASTER.stAlarms[1].aEventTexts[81] := '';
GVL_MASTER.stAlarms[1].aEventTexts[82] := '';

GVL_MASTER.stAlarms[1].aEventTexts[84] := '';
GVL_MASTER.stAlarms[1].aEventTexts[85] := '';
GVL_MASTER.stAlarms[1].aEventTexts[86] := '';
GVL_MASTER.stAlarms[1].aEventTexts[87] := ''; 
GVL_MASTER.stAlarms[1].aEventTexts[88] := '';
GVL_MASTER.stAlarms[1].aEventTexts[89] := '';

//Master Messages

GVL_MASTER.stAlarms[1].aEventTexts[100] := '';
GVL_MASTER.stAlarms[1].aEventTexts[101] := '';
GVL_MASTER.stAlarms[1].aEventTexts[102] := '';
GVL_MASTER.stAlarms[1].aEventTexts[103] := '';
GVL_MASTER.stAlarms[1].aEventTexts[104] := '';
GVL_MASTER.stAlarms[1].aEventTexts[105] := '';
GVL_MASTER.stAlarms[1].aEventTexts[106] := '';
END_METHOD

END_PROGRAM

// ---- POUs/C_LeakTest/PRG_Fault_LeakTest.TcPOU
PROGRAM PRG_Fault_LeakTest
VAR
	


				i						: INT;
END_VAR
VAR_IN_OUT

  aAlarms  : ARRAY[0..3] OF ST_Events;
END_VAR

ACT_FaultTrig();

(************************************** Faults reset **********************************************)
IF   GVL_HMI_GLOBAL.bResetButton THEN 
	FOR i := 0 TO 127 DO
		GVL_MASTER.stAlarms[2].aEventFlags[i] := FALSE;
	END_FOR
END_IF
//===============================================================
//Initialize event texts on first scan
IF NOT GVL_MASTER.stAlarms[2].bEventTextsSet THEN
	SetEventTexts();
	GVL_MASTER.stAlarms[2].bEventTextsSet := TRUE;
END_IF


(***************************************************************************************************)
//Immediate fault
GVL_MASTER.stAlarms[2].bImmediateFault := FALSE;
FOR i := 0 TO 32DO
	GVL_MASTER.stAlarms[2].bImmediateFault := GVL_MASTER.stAlarms[2].bImmediateFault OR GVL_MASTER.stAlarms[2].aEventFlags[i];
END_FOR

//Cycle stop fault
GVL_MASTER.stAlarms[2].bCycleStopFault := FALSE;
FOR i := 33 TO 79 DO
	GVL_MASTER.stAlarms[2].bCycleStopFault := GVL_MASTER.stAlarms[2].bCycleStopFault OR GVL_MASTER.stAlarms[2].aEventFlags[i];
END_FOR
//Cycle stop Request
GVL_MASTER.stAlarms[2].bCycleStopRequest := FALSE;
FOR i := 80 TO 99 DO
	GVL_MASTER.stAlarms[2].bCycleStopRequest := GVL_MASTER.stAlarms[2].bCycleStopRequest OR GVL_MASTER.stAlarms[2].aEventFlags[i];
END_FOR

ACTION ACT_FaultTrig:
(**************************************************************************************************)
(**************************** Master Immediate Fault Stop *****************************************)
(**************************************************************************************************)
(* Copy Safety Immediate Stop Faults to Master Immediate Stop Faults *)
(* *)

